KUKA KRL program: ps_com_geo_c1.src, ps_com_geo_c1.dat

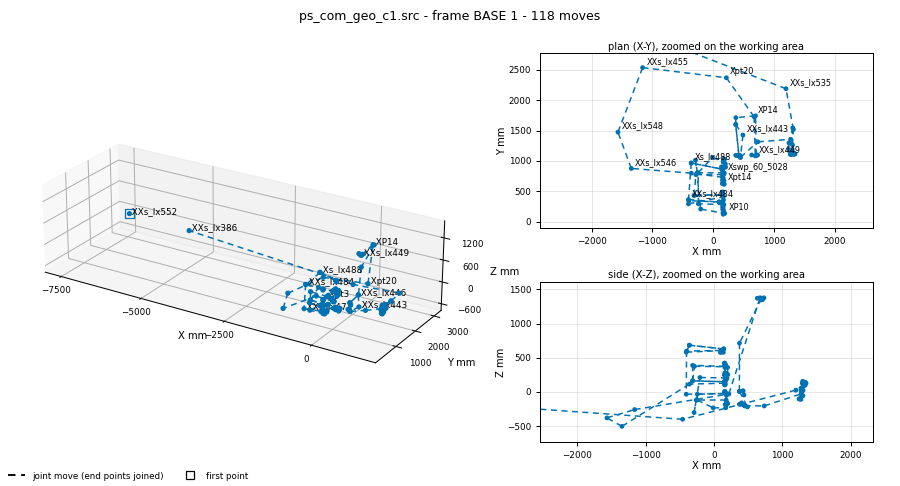
[picture p0: tool path of ps_com_geo_c1.src in frame BASE 1, 118 of 121 moves have a stored position in this frame; points joined in program order, loops and branches not executed]
--- ps_com_geo_c1.src ---
&ACCESS RVO1
&REL 24
&COMMENT Solda GUN C1 Geometria
&PARAM DISKPATH = KRC:\R1\Program\SOLDA LTC
DEF ps_com_geo_c1( )
;FOLD INI
;FOLD SPOTTECH INI
USERSPOT(#INIT)
;ENDFOLD (SPOTTECH INI)
  ;FOLD USER INI
    ;Make your modifications here

  ;ENDFOLD (USER INI)
;ENDFOLD (INI)

; Caracterização dos meios de produção:
; Versão Atual:
; 15/07/2013 12:00 Name: P13.050-R4 CHANGES: Geometria Actros
; LTA/LTB/MGS/MGSB/STB Pinça C1

chk_w1_wechs_ok ( )     ; CHECK FERRAMENTA: C1

;FOLD PTP Xs_lx552 CONT Vel=100 % PDAT57 Tool[1]:GUN_C1 Base[1]:ACTROS;%{PE}%R 8.2.20,%MKUKATPBASIS,%CMOVE,%VPTP,%P 1:PTP, 2:Xs_lx552, 3:C_DIS, 5:100, 7:PDAT57
$BWDSTART=FALSE
PDAT_ACT=PPDAT57
FDAT_ACT=FXs_lx552
BAS(#PTP_PARAMS,100)
PTP XXs_lx552 C_DIS
;ENDFOLD

if MaxStandMenge (1) then
  MaxStandmengeErreicht (1)
endif

IF (NOT(GHOST())) THEN
if Elektrodenwechsel (1) then
  e_Fraes1 ()
endif
ENDIF

;FOLD PTP c_lx33 CONT Vel=100 % P_OLP116 Tool[1]:GUN_C1 Base[1]:ACTROS;%{PE}%R 8.2.20,%MKUKATPBASIS,%CMOVE,%VPTP,%P 1:PTP, 2:c_lx33, 3:C_DIS, 5:100, 7:P_OLP116
$BWDSTART=FALSE
PDAT_ACT=PP_OLP116
FDAT_ACT=Fc_lx33
BAS(#PTP_PARAMS,100)
PTP Xc_lx33 C_DIS
;ENDFOLD
;FOLD PTP P3 CONT Vel=100 % PDAT59 Tool[1]:GUN_C1 Base[1]:ACTROS;%{PE}%R 8.2.20,%MKUKATPBASIS,%CMOVE,%VPTP,%P 1:PTP, 2:P3, 3:C_DIS, 5:100, 7:PDAT59
$BWDSTART=FALSE
PDAT_ACT=PPDAT59
FDAT_ACT=FP3
BAS(#PTP_PARAMS,100)
PTP XP3 C_DIS
;ENDFOLD
;FOLD PTP P2 Vel=100 % PDAT58 Tool[8]:TOOL_CHANGE Base[0];%{PE}%R 8.2.20,%MKUKATPBASIS,%CMOVE,%VPTP,%P 1:PTP, 2:P2, 3:, 5:100, 7:PDAT58
$BWDSTART=FALSE
PDAT_ACT=PPDAT58
FDAT_ACT=FP2
BAS(#PTP_PARAMS,100)
PTP XP2
;ENDFOLD

;FOLD OUT 3339 'R4 soldando' State=TRUE ;%{PE}%R 8.2.20,%MKUKATPBASIS,%COUT,%VOUTX,%P 2:3339, 3:R4 soldando, 5:TRUE, 6:
$OUT[3339]=TRUE
;ENDFOLD
;FOLD WAIT FOR ( IN 3339 'Aguarda lib solsar geometria' );%{PE}%R 8.2.20,%MKUKATPBASIS,%CEXT_WAIT_FOR,%VEXT_WAIT_FOR,%P 2:, 4:, 5:$IN, 6:3339, 7:Aguarda lib solsar geometria, 9:
WAIT FOR  ( $IN[3339] )
;ENDFOLD
;FOLD OUT 3339 'R4 soldando' State=FALSE ;%{PE}%R 8.2.20,%MKUKATPBASIS,%COUT,%VOUTX,%P 2:3339, 3:R4 soldando, 5:FALSE, 6:
$OUT[3339]=FALSE
;ENDFOLD
;FOLD OUT 3343 'R4 entregou peca Geo' State=FALSE ;%{PE}%R 8.2.20,%MKUKATPBASIS,%COUT,%VOUTX,%P 2:3343, 3:R4 entregou peca Geo, 5:FALSE, 6:
$OUT[3343]=FALSE
;ENDFOLD
;FOLD OUT 3348 'Fora area GEOBOX' State=FALSE ;%{PE}%R 8.2.20,%MKUKATPBASIS,%COUT,%VOUTX,%P 2:3348, 3:Fora area GEOBOX, 5:FALSE, 6:
$OUT[3348]=FALSE
;ENDFOLD
;FOLD  ;%{PE}%R 8.2.20,%MKUKATPBASIS,%CCOMMENT,%VNORMAL,%P 2:
;ENDFOLD
;FOLD Collision.Monitoring_5_On ;%{PE}%MKUKATPUSER
COLLSTOP( 5, 1 ) ;not Interrupt-Controlled
;ENDFOLD

;FOLD PTP Xs_lx488 CONT Vel=100 % P_OLP5 Tool[1]:GUN_C1 Base[1]:ACTROS;%{PE}%R8.2,%MKUKATPBASIS,%CMOVE,%VPTP,%P 1:PTP, 2:Xs_lx488, 3:C_DIS, 5:100, 7:P_OLP5
$BWDSTART = FALSE
PDAT_ACT= PP_OLP5
FDAT_ACT= Fs_lx488
BAS(#PTP_PARAMS,100)
PTP Xs_lx488 C_DIS
;ENDFOLD
;FOLD PTP Xs_lx487 CONT Vel=100 % PDAT2 Tool[1]:GUN_C1 Base[1]:ACTROS;%{PE}%R 8.2.19,%MKUKATPBASIS,%CMOVE,%VPTP,%P 1:PTP, 2:Xs_lx487, 3:C_DIS, 5:100, 7:PDAT2
$BWDSTART=FALSE
PDAT_ACT=PPDAT2
FDAT_ACT=FXs_lx487
BAS(#PTP_PARAMS,100)
PTP XXs_lx487 C_DIS
;ENDFOLD

;FOLD ; swp_60_5140;%{PE}%R 5.4.33,%MKUKATPBASIS,%CCOMMENT,%VNORMAL,%P 2:swp_60_5140
;ENDFOLD
;FOLD PTP swp_60_5140 P_OLP7 SPOT Gun=1 RETR CLS PgNo1=14 ACTIVE=1 Tool[1]:GUN_C1 Base[1]:ACTROS;%{PE}%R 8.2.2,%MKUKATPSPOT,%CSPOT,%VPTP,%P 1:PTP, 2:swp_60_5140, 3:, 5:100, 7:P_OLP7, 10:1, 12:#FIRST, 14:#CLO, 16:14, 18:1, 20:1, 22:0, 24:1, 25:S_OLP1
$BWDSTART=FALSE
PDAT_ACT=PP_OLP7
FDAT_ACT=Fswp_60_5140
BAS(#PTP_PARAMS,PP_OLP7.VEL)
S_ACT.GUN=1
S_ACT.PAIR=SDEFAULT.PAIR
S_ACT.RETR=#CLO
S_ACT.CLO_TM=1
S_ACT.PGNO1=14
S_ACT.PGNO2=SDEFAULT.PGNO2
S_ACT.PRESS1=SDEFAULT.PRESS1
S_ACT.PRESS2=SDEFAULT.PRESS2
S_READY=FALSE
PTP Xswp_60_5140
USERSPOT(#SPOT, S_ACT)
WAIT FOR S_READY
;ENDFOLD

;FOLD PTP Xs_lx502 CONT Vel=100 % PDAT6 Tool[1]:GUN_C1 Base[1]:ACTROS;%{PE}%R 8.2.20,%MKUKATPBASIS,%CMOVE,%VPTP,%P 1:PTP, 2:Xs_lx502, 3:C_DIS, 5:100, 7:PDAT6
$BWDSTART=FALSE
PDAT_ACT=PPDAT6
FDAT_ACT=FXs_lx502
BAS(#PTP_PARAMS,100)
PTP XXs_lx502 C_DIS
;ENDFOLD
;FOLD PTP Xs_lx486 CONT Vel=100 % P_OLP9 Tool[1]:GUN_C1 Base[1]:ACTROS;%{PE}%R8.2,%MKUKATPBASIS,%CMOVE,%VPTP,%P 1:PTP, 2:Xs_lx486, 3:C_DIS, 5:100, 7:P_OLP9
$BWDSTART = FALSE
PDAT_ACT= PP_OLP9
FDAT_ACT= Fs_lx486
BAS(#PTP_PARAMS,100)
PTP Xs_lx486 C_DIS
;ENDFOLD
;FOLD  ;%{PE}%R 8.2.20,%MKUKATPBASIS,%CCOMMENT,%VNORMAL,%P 2:
;ENDFOLD
;FOLD Collision.Monitoring_5_Off . ;%{PE}%MKUKATPUSER
COLLSTOP( 5, 2+0 )
;ENDFOLD

;FOLD PTP Xs_lx484 CONT Vel=100 % P_OLP10 Tool[1]:GUN_C1 Base[1]:ACTROS;%{PE}%R 8.2.20,%MKUKATPBASIS,%CMOVE,%VPTP,%P 1:PTP, 2:Xs_lx484, 3:C_DIS, 5:100, 7:P_OLP10
$BWDSTART=FALSE
PDAT_ACT=PP_OLP10
FDAT_ACT=FXs_lx484
BAS(#PTP_PARAMS,100)
PTP XXs_lx484 C_DIS
;ENDFOLD
;FOLD PTP Xs_lx504 CONT Vel=100 % PDAT8 Tool[1]:GUN_C1 Base[1]:ACTROS;%{PE}%R 8.2.20,%MKUKATPBASIS,%CMOVE,%VPTP,%P 1:PTP, 2:Xs_lx504, 3:C_DIS, 5:100, 7:PDAT8
$BWDSTART=FALSE
PDAT_ACT=PPDAT8
FDAT_ACT=FXs_lx504
BAS(#PTP_PARAMS,100)
PTP XXs_lx504 C_DIS
;ENDFOLD

;FOLD ; swp_60_5118;%{PE}%R 5.4.33,%MKUKATPBASIS,%CCOMMENT,%VNORMAL,%P 2:swp_60_5118
;ENDFOLD
;FOLD PTP swp_60_5118 P_OLP12 SPOT Gun=1 RETR CLS PgNo1=15 ACTIVE=1 Tool[1]:GUN_C1 Base[1]:ACTROS;%{PE}%R 8.2.2,%MKUKATPSPOT,%CSPOT,%VPTP,%P 1:PTP, 2:swp_60_5118, 3:, 5:100, 7:P_OLP12, 10:1, 12:#FIRST, 14:#CLO, 16:15, 18:1, 20:1, 22:0, 24:1, 25:S_OLP2
$BWDSTART=FALSE
PDAT_ACT=PP_OLP12
FDAT_ACT=Fswp_60_5118
BAS(#PTP_PARAMS,PP_OLP12.VEL)
S_ACT.GUN=1
S_ACT.PAIR=SDEFAULT.PAIR
S_ACT.RETR=#CLO
S_ACT.CLO_TM=1
S_ACT.PGNO1=15
S_ACT.PGNO2=SDEFAULT.PGNO2
S_ACT.PRESS1=SDEFAULT.PRESS1
S_ACT.PRESS2=SDEFAULT.PRESS2
S_READY=FALSE
PTP Xswp_60_5118
USERSPOT(#SPOT, S_ACT)
WAIT FOR S_READY
;ENDFOLD

;FOLD PTP Xs_lx506 CONT Vel=100 % PDAT10 Tool[1]:GUN_C1 Base[1]:ACTROS;%{PE}%R 8.2.20,%MKUKATPBASIS,%CMOVE,%VPTP,%P 1:PTP, 2:Xs_lx506, 3:C_DIS, 5:100, 7:PDAT10
$BWDSTART=FALSE
PDAT_ACT=PPDAT10
FDAT_ACT=FXs_lx506
BAS(#PTP_PARAMS,100)
PTP XXs_lx506 C_DIS
;ENDFOLD
;FOLD PTP Xs_lx482 CONT Vel=100 % P_OLP14 Tool[1]:GUN_C1 Base[1]:ACTROS;%{PE}%R 8.2.20,%MKUKATPBASIS,%CMOVE,%VPTP,%P 1:PTP, 2:Xs_lx482, 3:C_DIS, 5:100, 7:P_OLP14
$BWDSTART=FALSE
PDAT_ACT=PP_OLP14
FDAT_ACT=FXs_lx482
BAS(#PTP_PARAMS,100)
PTP XXs_lx482 C_DIS
;ENDFOLD
;FOLD PTP Xs_lx472 CONT Vel=100 % P_OLP16 Tool[1]:GUN_C1 Base[1]:ACTROS;%{PE}%R 8.2.20,%MKUKATPBASIS,%CMOVE,%VPTP,%P 1:PTP, 2:Xs_lx472, 3:C_DIS, 5:100, 7:P_OLP16
$BWDSTART=FALSE
PDAT_ACT=PP_OLP16
FDAT_ACT=FXs_lx472
BAS(#PTP_PARAMS,100)
PTP XXs_lx472 C_DIS
;ENDFOLD

;FOLD Collision.Monitoring_3_On ;%{PE}%MKUKATPUSER
COLLSTOP( 3, 1 ) ;Interrupt-Controlled
;ENDFOLD

;FOLD PTP Xs_lx510 CONT Vel=100 % PDAT14 Tool[1]:GUN_C1 Base[1]:ACTROS;%{PE}%R 8.2.20,%MKUKATPBASIS,%CMOVE,%VPTP,%P 1:PTP, 2:Xs_lx510, 3:C_DIS, 5:100, 7:PDAT14
$BWDSTART=FALSE
PDAT_ACT=PPDAT14
FDAT_ACT=FXs_lx510
BAS(#PTP_PARAMS,100)
PTP XXs_lx510 C_DIS
;ENDFOLD

;FOLD ; swp_60_5026;%{PE}%R 5.4.33,%MKUKATPBASIS,%CCOMMENT,%VNORMAL,%P 2:swp_60_5026
;ENDFOLD
;FOLD PTP swp_60_5026 P_OLP18 SPOT Gun=1 RETR CLS PgNo1=16 ACTIVE=1 Tool[1]:GUN_C1 Base[1]:ACTROS;%{PE}%R 8.2.2,%MKUKATPSPOT,%CSPOT,%VPTP,%P 1:PTP, 2:swp_60_5026, 3:, 5:100, 7:P_OLP18, 10:1, 12:#FIRST, 14:#CLO, 16:16, 18:1, 20:1, 22:0, 24:1, 25:S_OLP3
$BWDSTART=FALSE
PDAT_ACT=PP_OLP18
FDAT_ACT=Fswp_60_5026
BAS(#PTP_PARAMS,PP_OLP18.VEL)
S_ACT.GUN=1
S_ACT.PAIR=SDEFAULT.PAIR
S_ACT.RETR=#CLO
S_ACT.CLO_TM=1
S_ACT.PGNO1=16
S_ACT.PGNO2=SDEFAULT.PGNO2
S_ACT.PRESS1=SDEFAULT.PRESS1
S_ACT.PRESS2=SDEFAULT.PRESS2
S_READY=FALSE
PTP Xswp_60_5026
USERSPOT(#SPOT, S_ACT)
WAIT FOR S_READY
;ENDFOLD

;FOLD ; swp_60_5020;%{PE}%R 5.4.33,%MKUKATPBASIS,%CCOMMENT,%VNORMAL,%P 2:swp_60_5020
;ENDFOLD
;FOLD PTP swp_60_5020 P_OLP19 SPOT Gun=1 RETR CLS PgNo1=17 ACTIVE=1 Tool[1]:GUN_C1 Base[1]:ACTROS;%{PE}%R 8.2.2,%MKUKATPSPOT,%CSPOT,%VPTP,%P 1:PTP, 2:swp_60_5020, 3:, 5:100, 7:P_OLP19, 10:1, 12:#FIRST, 14:#CLO, 16:17, 18:1, 20:1, 22:0, 24:1, 25:S_OLP4
$BWDSTART=FALSE
PDAT_ACT=PP_OLP19
FDAT_ACT=Fswp_60_5020
BAS(#PTP_PARAMS,PP_OLP19.VEL)
S_ACT.GUN=1
S_ACT.PAIR=SDEFAULT.PAIR
S_ACT.RETR=#CLO
S_ACT.CLO_TM=1
S_ACT.PGNO1=17
S_ACT.PGNO2=SDEFAULT.PGNO2
S_ACT.PRESS1=SDEFAULT.PRESS1
S_ACT.PRESS2=SDEFAULT.PRESS2
S_READY=FALSE
PTP Xswp_60_5020
USERSPOT(#SPOT, S_ACT)
WAIT FOR S_READY
;ENDFOLD

;FOLD ; swp_60_5016;%{PE}%R 5.4.33,%MKUKATPBASIS,%CCOMMENT,%VNORMAL,%P 2:swp_60_5016
;ENDFOLD
;FOLD PTP swp_60_5016 P_OLP20 SPOT Gun=1 RETR CLS PgNo1=18 ACTIVE=1 Tool[1]:GUN_C1 Base[1]:ACTROS;%{PE}%R 8.2.2,%MKUKATPSPOT,%CSPOT,%VPTP,%P 1:PTP, 2:swp_60_5016, 3:, 5:100, 7:P_OLP20, 10:1, 12:#FIRST, 14:#CLO, 16:18, 18:1, 20:1, 22:0, 24:1, 25:S_OLP5
$BWDSTART=FALSE
PDAT_ACT=PP_OLP20
FDAT_ACT=Fswp_60_5016
BAS(#PTP_PARAMS,PP_OLP20.VEL)
S_ACT.GUN=1
S_ACT.PAIR=SDEFAULT.PAIR
S_ACT.RETR=#CLO
S_ACT.CLO_TM=1
S_ACT.PGNO1=18
S_ACT.PGNO2=SDEFAULT.PGNO2
S_ACT.PRESS1=SDEFAULT.PRESS1
S_ACT.PRESS2=SDEFAULT.PRESS2
S_READY=FALSE
PTP Xswp_60_5016
USERSPOT(#SPOT, S_ACT)
WAIT FOR S_READY
;ENDFOLD

;FOLD ; swp_60_5014;%{PE}%R 5.4.33,%MKUKATPBASIS,%CCOMMENT,%VNORMAL,%P 2:swp_60_5014
;ENDFOLD
;FOLD PTP swp_60_5014 P_OLP21 SPOT Gun=1 RETR CLS PgNo1=19 ACTIVE=1 Tool[1]:GUN_C1 Base[1]:ACTROS;%{PE}%R 8.2.2,%MKUKATPSPOT,%CSPOT,%VPTP,%P 1:PTP, 2:swp_60_5014, 3:, 5:100, 7:P_OLP21, 10:1, 12:#FIRST, 14:#CLO, 16:19, 18:1, 20:1, 22:0, 24:1, 25:S_OLP6
$BWDSTART=FALSE
PDAT_ACT=PP_OLP21
FDAT_ACT=Fswp_60_5014
BAS(#PTP_PARAMS,PP_OLP21.VEL)
S_ACT.GUN=1
S_ACT.PAIR=SDEFAULT.PAIR
S_ACT.RETR=#CLO
S_ACT.CLO_TM=1
S_ACT.PGNO1=19
S_ACT.PGNO2=SDEFAULT.PGNO2
S_ACT.PRESS1=SDEFAULT.PRESS1
S_ACT.PRESS2=SDEFAULT.PRESS2
S_READY=FALSE
PTP Xswp_60_5014
USERSPOT(#SPOT, S_ACT)
WAIT FOR S_READY
;ENDFOLD

;FOLD PTP Xs_lx469 CONT Vel=100 % P_OLP22 Tool[1]:GUN_C1 Base[1]:ACTROS;%{PE}%R 8.2.19,%MKUKATPBASIS,%CMOVE,%VPTP,%P 1:PTP, 2:Xs_lx469, 3:C_DIS, 5:100, 7:P_OLP22
$BWDSTART=FALSE
PDAT_ACT=PP_OLP22
FDAT_ACT=FXs_lx469
BAS(#PTP_PARAMS,100)
PTP XXs_lx469 C_DIS
;ENDFOLD
;FOLD PTP Xs_lx470 CONT Vel=100 % P_OLP23 Tool[1]:GUN_C1 Base[1]:ACTROS;%{PE}%R8.2,%MKUKATPBASIS,%CMOVE,%VPTP,%P 1:PTP, 2:Xs_lx470, 3:C_DIS, 5:100, 7:P_OLP23
$BWDSTART = FALSE
PDAT_ACT= PP_OLP23
FDAT_ACT= Fs_lx470
BAS(#PTP_PARAMS,100)
PTP Xs_lx470 C_DIS
;ENDFOLD
;FOLD PTP Xs_lx468 Vel=100 % P_OLP24 Tool[1]:GUN_C1 Base[1]:ACTROS;%{PE}%R 8.2.20,%MKUKATPBASIS,%CMOVE,%VPTP,%P 1:PTP, 2:Xs_lx468, 3:, 5:100, 7:P_OLP24
$BWDSTART=FALSE
PDAT_ACT=PP_OLP24
FDAT_ACT=FXs_lx468
BAS(#PTP_PARAMS,100)
PTP XXs_lx468
;ENDFOLD

;FOLD Collision.Monitoring_3_Off . ;%{PE}%MKUKATPUSER
COLLSTOP( 3, 2+0 )
;ENDFOLD
;FOLD ;%{PE}%R 8.2.20,%MKUKATPBASIS,%CCOMMENT,%VNORMAL,%P 2:
;ENDFOLD
;FOLD PTP Xlx507 CONT Vel=100 % P_OLP25 Tool[1]:GUN_C1 Base[1]:ACTROS;%{PE}%R8.2,%MKUKATPBASIS,%CMOVE,%VPTP,%P 1:PTP, 2:Xlx507, 3:C_DIS, 5:100, 7:P_OLP25
$BWDSTART = FALSE
PDAT_ACT= PP_OLP25
FDAT_ACT= Flx507
BAS(#PTP_PARAMS,100)
PTP Xlx507 C_DIS
;ENDFOLD
;FOLD PTP Xs_lx467 CONT Vel=100 % P_OLP26 Tool[1]:GUN_C1 Base[1]:ACTROS;%{PE}%R 8.2.20,%MKUKATPBASIS,%CMOVE,%VPTP,%P 1:PTP, 2:Xs_lx467, 3:C_DIS, 5:100, 7:P_OLP26
$BWDSTART=FALSE
PDAT_ACT=PP_OLP26
FDAT_ACT=FXs_lx467
BAS(#PTP_PARAMS,100)
PTP XXs_lx467 C_DIS
;ENDFOLD

;FOLD ; swp_60_5042;%{PE}%R 5.4.33,%MKUKATPBASIS,%CCOMMENT,%VNORMAL,%P 2:swp_60_5042
;ENDFOLD
;FOLD PTP swp_60_5042 P_OLP27 SPOT Gun=1 RETR CLS PgNo1=20 ACTIVE=1 Tool[1]:GUN_C1 Base[1]:ACTROS;%{PE}%R 8.2.2,%MKUKATPSPOT,%CSPOT,%VPTP,%P 1:PTP, 2:swp_60_5042, 3:, 5:100, 7:P_OLP27, 10:1, 12:#FIRST, 14:#CLO, 16:20, 18:1, 20:1, 22:0, 24:1, 25:S_OLP7
$BWDSTART=FALSE
PDAT_ACT=PP_OLP27
FDAT_ACT=Fswp_60_5042
BAS(#PTP_PARAMS,PP_OLP27.VEL)
S_ACT.GUN=1
S_ACT.PAIR=SDEFAULT.PAIR
S_ACT.RETR=#CLO
S_ACT.CLO_TM=1
S_ACT.PGNO1=20
S_ACT.PGNO2=SDEFAULT.PGNO2
S_ACT.PRESS1=SDEFAULT.PRESS1
S_ACT.PRESS2=SDEFAULT.PRESS2
S_READY=FALSE
PTP Xswp_60_5042
USERSPOT(#SPOT, S_ACT)
WAIT FOR S_READY
;ENDFOLD

;FOLD PTP Xs_lx512 CONT Vel=100 % PDAT16 Tool[1]:GUN_C1 Base[1]:ACTROS;%{PE}%R 8.2.19,%MKUKATPBASIS,%CMOVE,%VPTP,%P 1:PTP, 2:Xs_lx512, 3:C_DIS, 5:100, 7:PDAT16
$BWDSTART=FALSE
PDAT_ACT=PPDAT16
FDAT_ACT=FXs_lx512
BAS(#PTP_PARAMS,100)
PTP XXs_lx512 C_DIS
;ENDFOLD

;FOLD ; swp_60_5040;%{PE}%R 5.4.33,%MKUKATPBASIS,%CCOMMENT,%VNORMAL,%P 2:swp_60_5040
;ENDFOLD
;FOLD PTP swp_60_5040 P_OLP28 SPOT Gun=1 RETR CLS PgNo1=21 ACTIVE=1 Tool[1]:GUN_C1 Base[1]:ACTROS;%{PE}%R 8.2.2,%MKUKATPSPOT,%CSPOT,%VPTP,%P 1:PTP, 2:swp_60_5040, 3:, 5:100, 7:P_OLP28, 10:1, 12:#FIRST, 14:#CLO, 16:21, 18:1, 20:1, 22:0, 24:1, 25:S_OLP8
$BWDSTART=FALSE
PDAT_ACT=PP_OLP28
FDAT_ACT=Fswp_60_5040
BAS(#PTP_PARAMS,PP_OLP28.VEL)
S_ACT.GUN=1
S_ACT.PAIR=SDEFAULT.PAIR
S_ACT.RETR=#CLO
S_ACT.CLO_TM=1
S_ACT.PGNO1=21
S_ACT.PGNO2=SDEFAULT.PGNO2
S_ACT.PRESS1=SDEFAULT.PRESS1
S_ACT.PRESS2=SDEFAULT.PRESS2
S_READY=FALSE
PTP Xswp_60_5040
USERSPOT(#SPOT, S_ACT)
WAIT FOR S_READY
;ENDFOLD

;FOLD ; swp_60_5038;%{PE}%R 5.4.33,%MKUKATPBASIS,%CCOMMENT,%VNORMAL,%P 2:swp_60_5038
;ENDFOLD
;FOLD PTP swp_60_5038 P_OLP29 SPOT Gun=1 RETR OPN PgNo1=22 ACTIVE=1 Tool[1]:GUN_C1 Base[1]:ACTROS;%{PE}%R 8.2.2,%MKUKATPSPOT,%CSPOT,%VPTP,%P 1:PTP, 2:swp_60_5038, 3:, 5:100, 7:P_OLP29, 10:1, 12:#FIRST, 14:#OPN, 16:22, 18:1, 20:1, 22:0, 24:1, 25:S_OLP9
$BWDSTART=FALSE
PDAT_ACT=PP_OLP29
FDAT_ACT=Fswp_60_5038
BAS(#PTP_PARAMS,PP_OLP29.VEL)
S_ACT.GUN=1
S_ACT.PAIR=SDEFAULT.PAIR
S_ACT.RETR=#OPN
S_ACT.CLO_TM=1
S_ACT.PGNO1=22
S_ACT.PGNO2=SDEFAULT.PGNO2
S_ACT.PRESS1=SDEFAULT.PRESS1
S_ACT.PRESS2=SDEFAULT.PRESS2
S_READY=FALSE
PTP Xswp_60_5038
USERSPOT(#SPOT, S_ACT)
WAIT FOR S_READY
;ENDFOLD

;FOLD PTP Xs_lx514 CONT Vel=100 % PDAT18 Tool[1]:GUN_C1 Base[1]:ACTROS;%{PE}%R 8.2.19,%MKUKATPBASIS,%CMOVE,%VPTP,%P 1:PTP, 2:Xs_lx514, 3:C_DIS, 5:100, 7:PDAT18
$BWDSTART=FALSE
PDAT_ACT=PPDAT18
FDAT_ACT=FXs_lx514
BAS(#PTP_PARAMS,100)
PTP XXs_lx514 C_DIS
;ENDFOLD

;FOLD ; swp_60_5036;%{PE}%R 5.4.33,%MKUKATPBASIS,%CCOMMENT,%VNORMAL,%P 2:swp_60_5036
;ENDFOLD
;FOLD PTP swp_60_5036 PDAT45 SPOT Gun=1 RETR CLS PgNo1=23 ACTIVE=1 Tool[1]:GUN_C1 Base[1]:ACTROS;%{PE}%R 8.2.2,%MKUKATPSPOT,%CSPOT,%VPTP,%P 1:PTP, 2:swp_60_5036, 3:, 5:100, 7:PDAT45, 10:1, 12:#FIRST, 14:#CLO, 16:23, 18:1, 20:1, 22:0, 24:1, 25:S_OLP10
$BWDSTART=FALSE
PDAT_ACT=PPDAT45
FDAT_ACT=Fswp_60_5036
BAS(#PTP_PARAMS,PPDAT45.VEL)
S_ACT.GUN=1
S_ACT.PAIR=SDEFAULT.PAIR
S_ACT.RETR=#CLO
S_ACT.CLO_TM=1
S_ACT.PGNO1=23
S_ACT.PGNO2=SDEFAULT.PGNO2
S_ACT.PRESS1=SDEFAULT.PRESS1
S_ACT.PRESS2=SDEFAULT.PRESS2
S_READY=FALSE
PTP Xswp_60_5036
USERSPOT(#SPOT, S_ACT)
WAIT FOR S_READY
;ENDFOLD

;FOLD ; swp_60_5028;%{PE}%R 8.2.20,%MKUKATPBASIS,%CCOMMENT,%VNORMAL,%P 2:swp_60_5028
;ENDFOLD
;FOLD PTP swp_60_5028 P_OLP32 SPOT Gun=1 RETR CLS PgNo1=24 ACTIVE=1 Tool[1]:GUN_C1 Base[1]:ACTROS;%{PE}%R 8.2.2,%MKUKATPSPOT,%CSPOT,%VPTP,%P 1:PTP, 2:swp_60_5028, 3:, 5:100, 7:P_OLP32, 10:1, 12:#FIRST, 14:#CLO, 16:24, 18:1, 20:1, 22:0, 24:1, 25:S_OLP11
$BWDSTART=FALSE
PDAT_ACT=PP_OLP32
FDAT_ACT=Fswp_60_5028
BAS(#PTP_PARAMS,PP_OLP32.VEL)
S_ACT.GUN=1
S_ACT.PAIR=SDEFAULT.PAIR
S_ACT.RETR=#CLO
S_ACT.CLO_TM=1
S_ACT.PGNO1=24
S_ACT.PGNO2=SDEFAULT.PGNO2
S_ACT.PRESS1=SDEFAULT.PRESS1
S_ACT.PRESS2=SDEFAULT.PRESS2
S_READY=FALSE
PTP Xswp_60_5028
USERSPOT(#SPOT, S_ACT)
WAIT FOR S_READY
;ENDFOLD

;FOLD PTP Xs_lx464 CONT Vel=100 % P_OLP33 Tool[1]:GUN_C1 Base[1]:ACTROS;%{PE}%R8.2,%MKUKATPBASIS,%CMOVE,%VPTP,%P 1:PTP, 2:Xs_lx464, 3:C_DIS, 5:100, 7:P_OLP33
$BWDSTART = FALSE
PDAT_ACT= PP_OLP33
FDAT_ACT= Fs_lx464
BAS(#PTP_PARAMS,100)
PTP Xs_lx464 C_DIS
;ENDFOLD
;FOLD PTP Xs_lx465 CONT Vel=100 % P_OLP34 Tool[1]:GUN_C1 Base[1]:ACTROS;%{PE}%R 8.2.19,%MKUKATPBASIS,%CMOVE,%VPTP,%P 1:PTP, 2:Xs_lx465, 3:C_DIS, 5:100, 7:P_OLP34
$BWDSTART=FALSE
PDAT_ACT=PP_OLP34
FDAT_ACT=FXs_lx465
BAS(#PTP_PARAMS,100)
PTP XXs_lx465 C_DIS
;ENDFOLD
;FOLD PTP P8 CONT Vel=100 % PDAT65 Tool[1]:GUN_C1 Base[1]:ACTROS;%{PE}%R 8.2.20,%MKUKATPBASIS,%CMOVE,%VPTP,%P 1:PTP, 2:P8, 3:C_DIS, 5:100, 7:PDAT65
$BWDSTART=FALSE
PDAT_ACT=PPDAT65
FDAT_ACT=FP8
BAS(#PTP_PARAMS,100)
PTP XP8 C_DIS
;ENDFOLD
;FOLD ;%{PE}%R 8.2.20,%MKUKATPBASIS,%CCOMMENT,%VNORMAL,%P 2:
;ENDFOLD
;FOLD Collision.Monitoring_AREA_6_On ;%{PE}%MKUKATPUSER
COLLSTOP( 12, 1 ) ;not Interrupt-Controlled
;ENDFOLD
;FOLD ;%{PE}%R 8.2.20,%MKUKATPBASIS,%CCOMMENT,%VNORMAL,%P 2:
;ENDFOLD
;FOLD PTP P9 CONT Vel=100 % PDAT66 Tool[1]:GUN_C1 Base[1]:ACTROS;%{PE}%R 8.2.20,%MKUKATPBASIS,%CMOVE,%VPTP,%P 1:PTP, 2:P9, 3:C_DIS, 5:100, 7:PDAT66
$BWDSTART=FALSE
PDAT_ACT=PPDAT66
FDAT_ACT=FP9
BAS(#PTP_PARAMS,100)
PTP XP9 C_DIS
;ENDFOLD
;FOLD PTP P10 CONT Vel=100 % PDAT67 Tool[1]:GUN_C1 Base[1]:ACTROS;%{PE}%R 8.2.20,%MKUKATPBASIS,%CMOVE,%VPTP,%P 1:PTP, 2:P10, 3:C_DIS, 5:100, 7:PDAT67
$BWDSTART=FALSE
PDAT_ACT=PPDAT67
FDAT_ACT=FP10
BAS(#PTP_PARAMS,100)
PTP XP10 C_DIS
;ENDFOLD

;FOLD ; swp_60_5218;%{PE}%R 8.2.20,%MKUKATPBASIS,%CCOMMENT,%VNORMAL,%P 2:swp_60_5218
;ENDFOLD
;FOLD PTP swp_60_5218 PDAT68 SPOT Gun=1 RETR CLS PgNo1=29 ACTIVE=1 Tool[1]:GUN_C1 Base[1]:ACTROS;%{PE}%R 8.2.2,%MKUKATPSPOT,%CSPOT,%VPTP,%P 1:PTP, 2:swp_60_5218, 3:, 5:100, 7:PDAT68, 10:1, 12:#FIRST, 14:#CLO, 16:29, 18:1, 20:0, 22:0, 24:1, 25:NORMAL
$BWDSTART=FALSE
PDAT_ACT=PPDAT68
FDAT_ACT=Fswp_60_5218
BAS(#PTP_PARAMS,PPDAT68.VEL)
S_ACT.GUN=1
S_ACT.PAIR=SDEFAULT.PAIR
S_ACT.RETR=#CLO
S_ACT.CLO_TM=1
S_ACT.PGNO1=29
S_ACT.PGNO2=SDEFAULT.PGNO2
S_ACT.PRESS1=SDEFAULT.PRESS1
S_ACT.PRESS2=SDEFAULT.PRESS2
S_READY=FALSE
PTP Xswp_60_5218
USERSPOT(#SPOT, S_ACT)
WAIT FOR S_READY
;ENDFOLD

;FOLD PTP P13 CONT Vel=100 % PDAT70 Tool[1]:GUN_C1 Base[1]:ACTROS;%{PE}%R 8.2.20,%MKUKATPBASIS,%CMOVE,%VPTP,%P 1:PTP, 2:P13, 3:C_DIS, 5:100, 7:PDAT70
$BWDSTART=FALSE
PDAT_ACT=PPDAT70
FDAT_ACT=FP13
BAS(#PTP_PARAMS,100)
PTP XP13 C_DIS
;ENDFOLD

;FOLD ; swp_60_5190;%{PE}%R 8.2.20,%MKUKATPBASIS,%CCOMMENT,%VNORMAL,%P 2:swp_60_5190
;ENDFOLD
;FOLD PTP swp_60_5190 PDAT71 SPOT Gun=1 RETR CLS PgNo1=28 ACTIVE=1 Tool[1]:GUN_C1 Base[1]:ACTROS;%{PE}%R 8.2.2,%MKUKATPSPOT,%CSPOT,%VPTP,%P 1:PTP, 2:swp_60_5190, 3:, 5:100, 7:PDAT71, 10:1, 12:#FIRST, 14:#CLO, 16:28, 18:1, 20:0, 22:0, 24:1, 25:NORMAL
$BWDSTART=FALSE
PDAT_ACT=PPDAT71
FDAT_ACT=Fswp_60_5190
BAS(#PTP_PARAMS,PPDAT71.VEL)
S_ACT.GUN=1
S_ACT.PAIR=SDEFAULT.PAIR
S_ACT.RETR=#CLO
S_ACT.CLO_TM=1
S_ACT.PGNO1=28
S_ACT.PGNO2=SDEFAULT.PGNO2
S_ACT.PRESS1=SDEFAULT.PRESS1
S_ACT.PRESS2=SDEFAULT.PRESS2
S_READY=FALSE
PTP Xswp_60_5190
USERSPOT(#SPOT, S_ACT)
WAIT FOR S_READY
;ENDFOLD

;FOLD PTP pt1 CONT Vel=100 % PDAT72 Tool[1]:GUN_C1 Base[1]:ACTROS;%{PE}%R 8.2.20,%MKUKATPBASIS,%CMOVE,%VPTP,%P 1:PTP, 2:pt1, 3:C_DIS, 5:100, 7:PDAT72
$BWDSTART=FALSE
PDAT_ACT=PPDAT72
FDAT_ACT=Fpt1
BAS(#PTP_PARAMS,100)
PTP Xpt1 C_DIS
;ENDFOLD

;FOLD ; swp_60_5195;%{PE}%R 8.2.20,%MKUKATPBASIS,%CCOMMENT,%VNORMAL,%P 2:swp_60_5195
;ENDFOLD
;FOLD PTP swp_60_5195 PDAT73 SPOT Gun=1 RETR CLS PgNo1=27 ACTIVE=1 Tool[1]:GUN_C1 Base[1]:ACTROS;%{PE}%R 8.2.2,%MKUKATPSPOT,%CSPOT,%VPTP,%P 1:PTP, 2:swp_60_5195, 3:, 5:100, 7:PDAT73, 10:1, 12:#FIRST, 14:#CLO, 16:27, 18:1, 20:0, 22:0, 24:1, 25:NORMAL
$BWDSTART=FALSE
PDAT_ACT=PPDAT73
FDAT_ACT=Fswp_60_5195
BAS(#PTP_PARAMS,PPDAT73.VEL)
S_ACT.GUN=1
S_ACT.PAIR=SDEFAULT.PAIR
S_ACT.RETR=#CLO
S_ACT.CLO_TM=1
S_ACT.PGNO1=27
S_ACT.PGNO2=SDEFAULT.PGNO2
S_ACT.PRESS1=SDEFAULT.PRESS1
S_ACT.PRESS2=SDEFAULT.PRESS2
S_READY=FALSE
PTP Xswp_60_5195
USERSPOT(#SPOT, S_ACT)
WAIT FOR S_READY
;ENDFOLD

;FOLD PTP pt2 CONT Vel=100 % PDAT74 Tool[1]:GUN_C1 Base[1]:ACTROS;%{PE}%R 8.2.20,%MKUKATPBASIS,%CMOVE,%VPTP,%P 1:PTP, 2:pt2, 3:C_DIS, 5:100, 7:PDAT74
$BWDSTART=FALSE
PDAT_ACT=PPDAT74
FDAT_ACT=Fpt2
BAS(#PTP_PARAMS,100)
PTP Xpt2 C_DIS
;ENDFOLD
;FOLD PTP pt3 CONT Vel=100 % PDAT75 Tool[1]:GUN_C1 Base[1]:ACTROS;%{PE}%R 8.2.20,%MKUKATPBASIS,%CMOVE,%VPTP,%P 1:PTP, 2:pt3, 3:C_DIS, 5:100, 7:PDAT75
$BWDSTART=FALSE
PDAT_ACT=PPDAT75
FDAT_ACT=Fpt3
BAS(#PTP_PARAMS,100)
PTP Xpt3 C_DIS
;ENDFOLD

;FOLD ; swp_60_5203;%{PE}%R 8.2.20,%MKUKATPBASIS,%CCOMMENT,%VNORMAL,%P 2:swp_60_5203
;ENDFOLD
;FOLD PTP swp_60_5203 PDAT76 SPOT Gun=1 RETR CLS PgNo1=26 ACTIVE=1 Tool[1]:GUN_C1 Base[1]:ACTROS;%{PE}%R 8.2.2,%MKUKATPSPOT,%CSPOT,%VPTP,%P 1:PTP, 2:swp_60_5203, 3:, 5:100, 7:PDAT76, 10:1, 12:#FIRST, 14:#CLO, 16:26, 18:1, 20:0, 22:0, 24:1, 25:NORMAL
$BWDSTART=FALSE
PDAT_ACT=PPDAT76
FDAT_ACT=Fswp_60_5203
BAS(#PTP_PARAMS,PPDAT76.VEL)
S_ACT.GUN=1
S_ACT.PAIR=SDEFAULT.PAIR
S_ACT.RETR=#CLO
S_ACT.CLO_TM=1
S_ACT.PGNO1=26
S_ACT.PGNO2=SDEFAULT.PGNO2
S_ACT.PRESS1=SDEFAULT.PRESS1
S_ACT.PRESS2=SDEFAULT.PRESS2
S_READY=FALSE
PTP Xswp_60_5203
USERSPOT(#SPOT, S_ACT)
WAIT FOR S_READY
;ENDFOLD

;FOLD PTP pt4 Vel=100 % PDAT77 Tool[1]:GUN_C1 Base[1]:ACTROS;%{PE}%R 8.2.20,%MKUKATPBASIS,%CMOVE,%VPTP,%P 1:PTP, 2:pt4, 3:, 5:100, 7:PDAT77
$BWDSTART=FALSE
PDAT_ACT=PPDAT77
FDAT_ACT=Fpt4
BAS(#PTP_PARAMS,100)
PTP Xpt4
;ENDFOLD
;FOLD PTP pt5 CONT Vel=100 % PDAT78 Tool[1]:GUN_C1 Base[1]:ACTROS;%{PE}%R 8.2.20,%MKUKATPBASIS,%CMOVE,%VPTP,%P 1:PTP, 2:pt5, 3:C_DIS, 5:100, 7:PDAT78
$BWDSTART=FALSE
PDAT_ACT=PPDAT78
FDAT_ACT=Fpt5
BAS(#PTP_PARAMS,100)
PTP Xpt5 C_DIS
;ENDFOLD
;FOLD PTP pt6 CONT Vel=100 % PDAT79 Tool[1]:GUN_C1 Base[1]:ACTROS;%{PE}%R 8.2.20,%MKUKATPBASIS,%CMOVE,%VPTP,%P 1:PTP, 2:pt6, 3:C_DIS, 5:100, 7:PDAT79
$BWDSTART=FALSE
PDAT_ACT=PPDAT79
FDAT_ACT=Fpt6
BAS(#PTP_PARAMS,100)
PTP Xpt6 C_DIS
;ENDFOLD
;FOLD PTP pt7 Vel=100 % PDAT80 Tool[1]:GUN_C1 Base[1]:ACTROS;%{PE}%R 8.2.20,%MKUKATPBASIS,%CMOVE,%VPTP,%P 1:PTP, 2:pt7, 3:, 5:100, 7:PDAT80
$BWDSTART=FALSE
PDAT_ACT=PPDAT80
FDAT_ACT=Fpt7
BAS(#PTP_PARAMS,100)
PTP Xpt7
;ENDFOLD

; swp_60_5209
;FOLD PTP swp_60_5209 PDAT81 SPOT Gun=1 RETR CLS PgNo1=25 ACTIVE=1 Tool[1]:GUN_C1 Base[1]:ACTROS;%{PE}%R 8.2.2,%MKUKATPSPOT,%CSPOT,%VPTP,%P 1:PTP, 2:swp_60_5209, 3:, 5:100, 7:PDAT81, 10:1, 12:#FIRST, 14:#CLO, 16:25, 18:1, 20:0, 22:0, 24:1, 25:NORMAL
$BWDSTART=FALSE
PDAT_ACT=PPDAT81
FDAT_ACT=Fswp_60_5209
BAS(#PTP_PARAMS,PPDAT81.VEL)
S_ACT.GUN=1
S_ACT.PAIR=SDEFAULT.PAIR
S_ACT.RETR=#CLO
S_ACT.CLO_TM=1
S_ACT.PGNO1=25
S_ACT.PGNO2=SDEFAULT.PGNO2
S_ACT.PRESS1=SDEFAULT.PRESS1
S_ACT.PRESS2=SDEFAULT.PRESS2
S_READY=FALSE
PTP Xswp_60_5209
USERSPOT(#SPOT, S_ACT)
WAIT FOR S_READY
;ENDFOLD

;FOLD PTP pt8 Vel=100 % PDAT82 Tool[1]:GUN_C1 Base[1]:ACTROS;%{PE}%R 8.2.20,%MKUKATPBASIS,%CMOVE,%VPTP,%P 1:PTP, 2:pt8, 3:, 5:100, 7:PDAT82
$BWDSTART=FALSE
PDAT_ACT=PPDAT82
FDAT_ACT=Fpt8
BAS(#PTP_PARAMS,100)
PTP Xpt8
;ENDFOLD
;FOLD PTP pt9 Vel=100 % PDAT83 Tool[1]:GUN_C1 Base[1]:ACTROS;%{PE}%R 8.2.20,%MKUKATPBASIS,%CMOVE,%VPTP,%P 1:PTP, 2:pt9, 3:, 5:100, 7:PDAT83
$BWDSTART=FALSE
PDAT_ACT=PPDAT83
FDAT_ACT=Fpt9
BAS(#PTP_PARAMS,100)
PTP Xpt9
;ENDFOLD
;FOLD PTP Xs_lx463 Vel=100 % P_OLP52 Tool[1]:GUN_C1 Base[1]:ACTROS;%{PE}%R 8.2.20,%MKUKATPBASIS,%CMOVE,%VPTP,%P 1:PTP, 2:Xs_lx463, 3:, 5:100, 7:P_OLP52
$BWDSTART=FALSE
PDAT_ACT=PP_OLP52
FDAT_ACT=FXs_lx463
BAS(#PTP_PARAMS,100)
PTP XXs_lx463
;ENDFOLD

;FOLD Collision.Monitoring_5_On ;%{PE}%MKUKATPUSER
COLLSTOP( 5, 1 ) ;not Interrupt-Controlled
;ENDFOLD
;FOLD Collision.Monitoring_AREA_6_Off . ;%{PE}%MKUKATPUSER
COLLSTOP( 12, 2+0 )
;ENDFOLD

;FOLD PTP Xs_lx464 CONT Vel=100 % P_OLP118 Tool[1]:GUN_C1 Base[1]:ACTROS;%{PE}%R 8.2.20,%MKUKATPBASIS,%CMOVE,%VPTP,%P 1:PTP, 2:Xs_lx464, 3:C_DIS, 5:100, 7:P_OLP118
$BWDSTART=FALSE
PDAT_ACT=PP_OLP118
FDAT_ACT=FXs_lx464
BAS(#PTP_PARAMS,100)
PTP XXs_lx464 C_DIS
;ENDFOLD

;FOLD ; swp_60_5096;%{PE}%R 8.2.20,%MKUKATPBASIS,%CCOMMENT,%VNORMAL,%P 2:swp_60_5096
;ENDFOLD
;FOLD PTP swp_60_5097 P_OLP119 SPOT Gun=1 RETR CLS PgNo1=32 ACTIVE=1 Tool[1]:GUN_C1 Base[1]:ACTROS;%{PE}%R 8.2.2,%MKUKATPSPOT,%CSPOT,%VPTP,%P 1:PTP, 2:swp_60_5097, 3:, 5:100, 7:P_OLP119, 10:1, 12:#FIRST, 14:#CLO, 16:32, 18:1, 20:1, 22:0, 24:1, 25:S_OLP19
$BWDSTART=FALSE
PDAT_ACT=PP_OLP119
FDAT_ACT=Fswp_60_5097
BAS(#PTP_PARAMS,PP_OLP119.VEL)
S_ACT.GUN=1
S_ACT.PAIR=SDEFAULT.PAIR
S_ACT.RETR=#CLO
S_ACT.CLO_TM=1
S_ACT.PGNO1=32
S_ACT.PGNO2=SDEFAULT.PGNO2
S_ACT.PRESS1=SDEFAULT.PRESS1
S_ACT.PRESS2=SDEFAULT.PRESS2
S_READY=FALSE
PTP Xswp_60_5097
USERSPOT(#SPOT, S_ACT)
WAIT FOR S_READY

;ENDFOLD

;FOLD ; swp_60_5098;%{PE}%R 8.2.20,%MKUKATPBASIS,%CCOMMENT,%VNORMAL,%P 2:swp_60_5098
;ENDFOLD
;FOLD PTP swp_60_5099 P_OLP120 SPOT Gun=1 RETR CLS PgNo1=31 ACTIVE=1 Tool[1]:GUN_C1 Base[1]:ACTROS;%{PE}%R 8.2.2,%MKUKATPSPOT,%CSPOT,%VPTP,%P 1:PTP, 2:swp_60_5099, 3:, 5:100, 7:P_OLP120, 10:1, 12:#FIRST, 14:#CLO, 16:31, 18:1, 20:1, 22:0, 24:1, 25:S_OLP18
$BWDSTART=FALSE
PDAT_ACT=PP_OLP120
FDAT_ACT=Fswp_60_5099
BAS(#PTP_PARAMS,PP_OLP120.VEL)
S_ACT.GUN=1
S_ACT.PAIR=SDEFAULT.PAIR
S_ACT.RETR=#CLO
S_ACT.CLO_TM=1
S_ACT.PGNO1=31
S_ACT.PGNO2=SDEFAULT.PGNO2
S_ACT.PRESS1=SDEFAULT.PRESS1
S_ACT.PRESS2=SDEFAULT.PRESS2
S_READY=FALSE
PTP Xswp_60_5099
USERSPOT(#SPOT, S_ACT)
WAIT FOR S_READY

;ENDFOLD

;FOLD ; swp_60_5100;%{PE}%R 8.2.20,%MKUKATPBASIS,%CCOMMENT,%VNORMAL,%P 2:swp_60_5100
;ENDFOLD
;FOLD PTP swp_60_5101 P_OLP121 SPOT Gun=1 RETR OPN PgNo1=30 ACTIVE=1 Tool[1]:GUN_C1 Base[1]:ACTROS;%{PE}%R 8.2.2,%MKUKATPSPOT,%CSPOT,%VPTP,%P 1:PTP, 2:swp_60_5101, 3:, 5:100, 7:P_OLP121, 10:1, 12:#FIRST, 14:#OPN, 16:30, 18:1, 20:1, 22:0, 24:1, 25:S_OLP17
$BWDSTART=FALSE
PDAT_ACT=PP_OLP121
FDAT_ACT=Fswp_60_5101
BAS(#PTP_PARAMS,PP_OLP121.VEL)
S_ACT.GUN=1
S_ACT.PAIR=SDEFAULT.PAIR
S_ACT.RETR=#OPN
S_ACT.CLO_TM=1
S_ACT.PGNO1=30
S_ACT.PGNO2=SDEFAULT.PGNO2
S_ACT.PRESS1=SDEFAULT.PRESS1
S_ACT.PRESS2=SDEFAULT.PRESS2
S_READY=FALSE
PTP Xswp_60_5101
USERSPOT(#SPOT, S_ACT)
WAIT FOR S_READY
;ENDFOLD

;FOLD PTP Xlx510 CONT Vel=100 % P_OLP59 Tool[1]:GUN_C1 Base[1]:ACTROS;%{PE}%R 8.2.20,%MKUKATPBASIS,%CMOVE,%VPTP,%P 1:PTP, 2:Xlx510, 3:C_DIS, 5:100, 7:P_OLP59
$BWDSTART=FALSE
PDAT_ACT=PP_OLP59
FDAT_ACT=FXlx510
BAS(#PTP_PARAMS,100)
PTP XXlx510 C_DIS
;ENDFOLD
;FOLD PTP Xlx511 CONT Vel=100 % P_OLP60 Tool[1]:GUN_C1 Base[1]:ACTROS;%{PE}%R 8.2.20,%MKUKATPBASIS,%CMOVE,%VPTP,%P 1:PTP, 2:Xlx511, 3:C_DIS, 5:100, 7:P_OLP60
$BWDSTART=FALSE
PDAT_ACT=PP_OLP60
FDAT_ACT=FXlx511
BAS(#PTP_PARAMS,100)
PTP XXlx511 C_DIS
;ENDFOLD

;FOLD ; swp_60_5084;%{PE}%R 8.2.20,%MKUKATPBASIS,%CCOMMENT,%VNORMAL,%P 2:swp_60_5084
;ENDFOLD
;FOLD PTP swp_60_5085 P_OLP122 SPOT Gun=1 RETR CLS PgNo1=35 ACTIVE=1 Tool[1]:GUN_C1 Base[1]:ACTROS;%{PE}%R 8.2.2,%MKUKATPSPOT,%CSPOT,%VPTP,%P 1:PTP, 2:swp_60_5085, 3:, 5:100, 7:P_OLP122, 10:1, 12:#FIRST, 14:#CLO, 16:35, 18:1, 20:1, 22:0, 24:1, 25:S_OLP22
$BWDSTART=FALSE
PDAT_ACT=PP_OLP122
FDAT_ACT=Fswp_60_5085
BAS(#PTP_PARAMS,PP_OLP122.VEL)
S_ACT.GUN=1
S_ACT.PAIR=SDEFAULT.PAIR
S_ACT.RETR=#CLO
S_ACT.CLO_TM=1
S_ACT.PGNO1=35
S_ACT.PGNO2=SDEFAULT.PGNO2
S_ACT.PRESS1=SDEFAULT.PRESS1
S_ACT.PRESS2=SDEFAULT.PRESS2
S_READY=FALSE
PTP Xswp_60_5085
USERSPOT(#SPOT, S_ACT)
WAIT FOR S_READY

;ENDFOLD

;FOLD PTP Xlx509 CONT Vel=100 % P_OLP61 Tool[1]:GUN_C1 Base[1]:ACTROS;%{PE}%R 8.2.20,%MKUKATPBASIS,%CMOVE,%VPTP,%P 1:PTP, 2:Xlx509, 3:C_DIS, 5:100, 7:P_OLP61
$BWDSTART=FALSE
PDAT_ACT=PP_OLP61
FDAT_ACT=FXlx509
BAS(#PTP_PARAMS,100)
PTP XXlx509 C_DIS
;ENDFOLD

;FOLD ; swp_60_5076;%{PE}%R 5.4.33,%MKUKATPBASIS,%CCOMMENT,%VNORMAL,%P 2:swp_60_5076
;ENDFOLD
;FOLD PTP swp_60_5076 P_OLP63 SPOT Gun=1 RETR OPN PgNo1=34 ACTIVE=1 Tool[1]:GUN_C1 Base[1]:ACTROS;%{PE}%R 8.2.2,%MKUKATPSPOT,%CSPOT,%VPTP,%P 1:PTP, 2:swp_60_5076, 3:, 5:100, 7:P_OLP63, 10:1, 12:#FIRST, 14:#OPN, 16:34, 18:1, 20:1, 22:0, 24:1, 25:S_OLP21
$BWDSTART=FALSE
PDAT_ACT=PP_OLP63
FDAT_ACT=Fswp_60_5076
BAS(#PTP_PARAMS,PP_OLP63.VEL)
S_ACT.GUN=1
S_ACT.PAIR=SDEFAULT.PAIR
S_ACT.RETR=#OPN
S_ACT.CLO_TM=1
S_ACT.PGNO1=34
S_ACT.PGNO2=SDEFAULT.PGNO2
S_ACT.PRESS1=SDEFAULT.PRESS1
S_ACT.PRESS2=SDEFAULT.PRESS2
S_READY=FALSE
PTP Xswp_60_5076
USERSPOT(#SPOT, S_ACT)
WAIT FOR S_READY
;ENDFOLD

;FOLD PTP pt11 CONT Vel=100 % PDAT85 Tool[1]:GUN_C1 Base[1]:ACTROS;%{PE}%R 8.2.20,%MKUKATPBASIS,%CMOVE,%VPTP,%P 1:PTP, 2:pt11, 3:C_DIS, 5:100, 7:PDAT85
$BWDSTART=FALSE
PDAT_ACT=PPDAT85
FDAT_ACT=Fpt11
BAS(#PTP_PARAMS,100)
PTP Xpt11 C_DIS
;ENDFOLD
;FOLD PTP pt12 CONT Vel=100 % PDAT86 Tool[1]:GUN_C1 Base[1]:ACTROS;%{PE}%R 8.2.20,%MKUKATPBASIS,%CMOVE,%VPTP,%P 1:PTP, 2:pt12, 3:C_DIS, 5:100, 7:PDAT86
$BWDSTART=FALSE
PDAT_ACT=PPDAT86
FDAT_ACT=Fpt12
BAS(#PTP_PARAMS,100)
PTP Xpt12 C_DIS
;ENDFOLD
;FOLD PTP pt13 CONT Vel=100 % PDAT87 Tool[1]:GUN_C1 Base[1]:ACTROS;%{PE}%R 8.2.20,%MKUKATPBASIS,%CMOVE,%VPTP,%P 1:PTP, 2:pt13, 3:C_DIS, 5:100, 7:PDAT87
$BWDSTART=FALSE
PDAT_ACT=PPDAT87
FDAT_ACT=Fpt13
BAS(#PTP_PARAMS,100)
PTP Xpt13 C_DIS
;ENDFOLD
;FOLD PTP pt14 Vel=100 % PDAT88 Tool[1]:GUN_C1 Base[1]:ACTROS;%{PE}%R 8.2.20,%MKUKATPBASIS,%CMOVE,%VPTP,%P 1:PTP, 2:pt14, 3:, 5:100, 7:PDAT88
$BWDSTART=FALSE
PDAT_ACT=PPDAT88
FDAT_ACT=Fpt14
BAS(#PTP_PARAMS,100)
PTP Xpt14
;ENDFOLD

;FOLD ; swp_60_5066;%{PE}%R 8.2.20,%MKUKATPBASIS,%CCOMMENT,%VNORMAL,%P 2:swp_60_5066
;ENDFOLD
;FOLD PTP swp_60_5066 PDAT89 SPOT Gun=1 RETR OPN PgNo1=48 ACTIVE=1 Tool[1]:GUN_C1 Base[1]:ACTROS;%{PE}%R 8.2.2,%MKUKATPSPOT,%CSPOT,%VPTP,%P 1:PTP, 2:swp_60_5066, 3:, 5:100, 7:PDAT89, 10:1, 12:#FIRST, 14:#OPN, 16:48, 18:1, 20:0, 22:0, 24:1, 25:NORMAL
$BWDSTART=FALSE
PDAT_ACT=PPDAT89
FDAT_ACT=Fswp_60_5066
BAS(#PTP_PARAMS,PPDAT89.VEL)
S_ACT.GUN=1
S_ACT.PAIR=SDEFAULT.PAIR
S_ACT.RETR=#OPN
S_ACT.CLO_TM=1
S_ACT.PGNO1=48
S_ACT.PGNO2=SDEFAULT.PGNO2
S_ACT.PRESS1=SDEFAULT.PRESS1
S_ACT.PRESS2=SDEFAULT.PRESS2
S_READY=FALSE
PTP Xswp_60_5066
USERSPOT(#SPOT, S_ACT)
WAIT FOR S_READY
;ENDFOLD

;FOLD PTP pt15 Vel=100 % PDAT90 Tool[1]:GUN_C1 Base[1]:ACTROS;%{PE}%R 8.2.20,%MKUKATPBASIS,%CMOVE,%VPTP,%P 1:PTP, 2:pt15, 3:, 5:100, 7:PDAT90
$BWDSTART=FALSE
PDAT_ACT=PPDAT90
FDAT_ACT=Fpt15
BAS(#PTP_PARAMS,100)
PTP Xpt15
;ENDFOLD
;FOLD PTP pt16 CONT Vel=100 % PDAT91 Tool[1]:GUN_C1 Base[1]:ACTROS;%{PE}%R 8.2.20,%MKUKATPBASIS,%CMOVE,%VPTP,%P 1:PTP, 2:pt16, 3:C_DIS, 5:100, 7:PDAT91
$BWDSTART=FALSE
PDAT_ACT=PPDAT91
FDAT_ACT=Fpt16
BAS(#PTP_PARAMS,100)
PTP Xpt16 C_DIS
;ENDFOLD
;FOLD PTP pt18 CONT Vel=100 % PDAT93 Tool[1]:GUN_C1 Base[1]:ACTROS;%{PE}%R 8.2.20,%MKUKATPBASIS,%CMOVE,%VPTP,%P 1:PTP, 2:pt18, 3:C_DIS, 5:100, 7:PDAT93
$BWDSTART=FALSE
PDAT_ACT=PPDAT93
FDAT_ACT=Fpt18
BAS(#PTP_PARAMS,100)
PTP Xpt18 C_DIS
;ENDFOLD
;FOLD PTP pt19 CONT Vel=100 % PDAT94 Tool[1]:GUN_C1 Base[1]:ACTROS;%{PE}%R 8.2.20,%MKUKATPBASIS,%CMOVE,%VPTP,%P 1:PTP, 2:pt19, 3:C_DIS, 5:100, 7:PDAT94
$BWDSTART=FALSE
PDAT_ACT=PPDAT94
FDAT_ACT=Fpt19
BAS(#PTP_PARAMS,100)
PTP Xpt19 C_DIS
;ENDFOLD

;FOLD PTP Xs_lx456 CONT Vel=100 % P_OLP64 Tool[1]:GUN_C1 Base[1]:ACTROS;%{PE}%R 8.2.20,%MKUKATPBASIS,%CMOVE,%VPTP,%P 1:PTP, 2:Xs_lx456, 3:C_DIS, 5:100, 7:P_OLP64
$BWDSTART=FALSE
PDAT_ACT=PP_OLP64
FDAT_ACT=FXs_lx456
BAS(#PTP_PARAMS,100)
PTP XXs_lx456 C_DIS
;ENDFOLD

;FOLD Collision.Monitoring_5_Off . ;%{PE}%MKUKATPUSER
COLLSTOP( 5, 2+0 )
;ENDFOLD

;FOLD PTP Xs_lx546 CONT Vel=100 % PDAT51 Tool[1]:GUN_C1 Base[1]:ACTROS;%{PE}%R 8.2.20,%MKUKATPBASIS,%CMOVE,%VPTP,%P 1:PTP, 2:Xs_lx546, 3:C_DIS, 5:100, 7:PDAT51
$BWDSTART=FALSE
PDAT_ACT=PPDAT51
FDAT_ACT=FXs_lx546
BAS(#PTP_PARAMS,100)
PTP XXs_lx546 C_DIS
;ENDFOLD
;FOLD PTP Xs_lx548 Vel=100 % PDAT53 Tool[1]:GUN_C1 Base[1]:ACTROS;%{PE}%R 8.2.20,%MKUKATPBASIS,%CMOVE,%VPTP,%P 1:PTP, 2:Xs_lx548, 3:, 5:100, 7:PDAT53
$BWDSTART=FALSE
PDAT_ACT=PPDAT53
FDAT_ACT=FXs_lx548
BAS(#PTP_PARAMS,100)
PTP XXs_lx548
;ENDFOLD
;FOLD PTP Xs_lx455 CONT Vel=100 % P_OLP69 Tool[1]:GUN_C1 Base[1]:ACTROS;%{PE}%R 8.2.19,%MKUKATPBASIS,%CMOVE,%VPTP,%P 1:PTP, 2:Xs_lx455, 3:C_DIS, 5:100, 7:P_OLP69
$BWDSTART=FALSE
PDAT_ACT=PP_OLP69
FDAT_ACT=FXs_lx455
BAS(#PTP_PARAMS,100)
PTP XXs_lx455 C_DIS
;ENDFOLD
;FOLD  ;%{PE}%R 8.2.20,%MKUKATPBASIS,%CCOMMENT,%VNORMAL,%P 2:
;ENDFOLD
;FOLD Collision.Monitoring_2_On ;%{PE}%MKUKATPUSER
COLLSTOP( 2, 1 ) ;Interrupt-Controlled
;ENDFOLD
;FOLD  ;%{PE}%R 8.2.20,%MKUKATPBASIS,%CCOMMENT,%VNORMAL,%P 2:
;ENDFOLD
;FOLD PTP pt20 CONT Vel=100 % PDAT95 Tool[1]:GUN_C1 Base[1]:ACTROS;%{PE}%R 8.2.20,%MKUKATPBASIS,%CMOVE,%VPTP,%P 1:PTP, 2:pt20, 3:C_DIS, 5:100, 7:PDAT95
$BWDSTART=FALSE
PDAT_ACT=PPDAT95
FDAT_ACT=Fpt20
BAS(#PTP_PARAMS,100)
PTP Xpt20 C_DIS
;ENDFOLD
;FOLD PTP P14 CONT Vel=100 % PDAT96 Tool[1]:GUN_C1 Base[1]:ACTROS;%{PE}%R 8.2.20,%MKUKATPBASIS,%CMOVE,%VPTP,%P 1:PTP, 2:P14, 3:C_DIS, 5:100, 7:PDAT96
$BWDSTART=FALSE
PDAT_ACT=PPDAT96
FDAT_ACT=FP14
BAS(#PTP_PARAMS,100)
PTP XP14 C_DIS
;ENDFOLD
;FOLD PTP Xs_lx449 CONT Vel=100 % P_OLP72 Tool[1]:GUN_C1 Base[1]:ACTROS;%{PE}%R 8.2.19,%MKUKATPBASIS,%CMOVE,%VPTP,%P 1:PTP, 2:Xs_lx449, 3:C_DIS, 5:100, 7:P_OLP72
$BWDSTART=FALSE
PDAT_ACT=PP_OLP72
FDAT_ACT=FXs_lx449
BAS(#PTP_PARAMS,100)
PTP XXs_lx449 C_DIS
;ENDFOLD

;FOLD ; swp_60_5626;%{PE}%R 5.4.33,%MKUKATPBASIS,%CCOMMENT,%VNORMAL,%P 2:swp_60_5626
;ENDFOLD
;FOLD PTP swp_60_5626 P_OLP73 SPOT Gun=1 RETR CLS PgNo1=36 ACTIVE=1 Tool[1]:GUN_C1 Base[1]:ACTROS;%{PE}%R 8.2.2,%MKUKATPSPOT,%CSPOT,%VPTP,%P 1:PTP, 2:swp_60_5626, 3:, 5:100, 7:P_OLP73, 10:1, 12:#FIRST, 14:#CLO, 16:36, 18:1, 20:1, 22:0, 24:1, 25:S_OLP23
$BWDSTART=FALSE
PDAT_ACT=PP_OLP73
FDAT_ACT=Fswp_60_5626
BAS(#PTP_PARAMS,PP_OLP73.VEL)
S_ACT.GUN=1
S_ACT.PAIR=SDEFAULT.PAIR
S_ACT.RETR=#CLO
S_ACT.CLO_TM=1
S_ACT.PGNO1=36
S_ACT.PGNO2=SDEFAULT.PGNO2
S_ACT.PRESS1=SDEFAULT.PRESS1
S_ACT.PRESS2=SDEFAULT.PRESS2
S_READY=FALSE
PTP Xswp_60_5626
USERSPOT(#SPOT, S_ACT)
WAIT FOR S_READY
;ENDFOLD

;FOLD ; swp_60_5640;%{PE}%R 5.4.33,%MKUKATPBASIS,%CCOMMENT,%VNORMAL,%P 2:swp_60_5640
;ENDFOLD
;FOLD PTP swp_60_5640 P_OLP74 SPOT Gun=1 RETR CLS PgNo1=37 ACTIVE=1 Tool[1]:GUN_C1 Base[1]:ACTROS;%{PE}%R 8.2.2,%MKUKATPSPOT,%CSPOT,%VPTP,%P 1:PTP, 2:swp_60_5640, 3:, 5:100, 7:P_OLP74, 10:1, 12:#FIRST, 14:#CLO, 16:37, 18:1, 20:1, 22:0, 24:1, 25:S_OLP24
$BWDSTART=FALSE
PDAT_ACT=PP_OLP74
FDAT_ACT=Fswp_60_5640
BAS(#PTP_PARAMS,PP_OLP74.VEL)
S_ACT.GUN=1
S_ACT.PAIR=SDEFAULT.PAIR
S_ACT.RETR=#CLO
S_ACT.CLO_TM=1
S_ACT.PGNO1=37
S_ACT.PGNO2=SDEFAULT.PGNO2
S_ACT.PRESS1=SDEFAULT.PRESS1
S_ACT.PRESS2=SDEFAULT.PRESS2
S_READY=FALSE
PTP Xswp_60_5640
USERSPOT(#SPOT, S_ACT)
WAIT FOR S_READY
;ENDFOLD

;FOLD PTP Xs_lx447 CONT Vel=100 % P_OLP75 Tool[1]:GUN_C1 Base[1]:ACTROS;%{PE}%R 8.2.19,%MKUKATPBASIS,%CMOVE,%VPTP,%P 1:PTP, 2:Xs_lx447, 3:C_DIS, 5:100, 7:P_OLP75
$BWDSTART=FALSE
PDAT_ACT=PP_OLP75
FDAT_ACT=FXs_lx447
BAS(#PTP_PARAMS,100)
PTP XXs_lx447 C_DIS
;ENDFOLD
;FOLD PTP Xs_lx448 CONT Vel=100 % P_OLP76 Tool[1]:GUN_C1 Base[1]:ACTROS;%{PE}%R 8.2.19,%MKUKATPBASIS,%CMOVE,%VPTP,%P 1:PTP, 2:Xs_lx448, 3:C_DIS, 5:100, 7:P_OLP76
$BWDSTART=FALSE
PDAT_ACT=PP_OLP76
FDAT_ACT=FXs_lx448
BAS(#PTP_PARAMS,100)
PTP XXs_lx448 C_DIS
;ENDFOLD
;FOLD PTP P15 CONT Vel=100 % PDAT97 Tool[1]:GUN_C1 Base[1]:ACTROS;%{PE}%R 8.2.20,%MKUKATPBASIS,%CMOVE,%VPTP,%P 1:PTP, 2:P15, 3:C_DIS, 5:100, 7:PDAT97
$BWDSTART=FALSE
PDAT_ACT=PPDAT97
FDAT_ACT=FP15
BAS(#PTP_PARAMS,100)
PTP XP15 C_DIS
;ENDFOLD

;FOLD PTP Xs_lx446 CONT Vel=100 % P_OLP77 Tool[1]:GUN_C1 Base[1]:ACTROS;%{PE}%R 8.2.20,%MKUKATPBASIS,%CMOVE,%VPTP,%P 1:PTP, 2:Xs_lx446, 3:C_DIS, 5:100, 7:P_OLP77
$BWDSTART=FALSE
PDAT_ACT=PP_OLP77
FDAT_ACT=FXs_lx446
BAS(#PTP_PARAMS,100)
PTP XXs_lx446 C_DIS
;ENDFOLD
;FOLD PTP Xs_lx445 CONT Vel=100 % P_OLP78 Tool[1]:GUN_C1 Base[1]:ACTROS;%{PE}%R 8.2.20,%MKUKATPBASIS,%CMOVE,%VPTP,%P 1:PTP, 2:Xs_lx445, 3:C_DIS, 5:100, 7:P_OLP78
$BWDSTART=FALSE
PDAT_ACT=PP_OLP78
FDAT_ACT=FXs_lx445
BAS(#PTP_PARAMS,100)
PTP XXs_lx445 C_DIS
;ENDFOLD

;FOLD ; swp_60_5060;%{PE}%R 5.4.33,%MKUKATPBASIS,%CCOMMENT,%VNORMAL,%P 2:swp_60_5060
;ENDFOLD
;FOLD PTP swp_60_5060 P_OLP79 SPOT Gun=1 RETR CLS PgNo1=38 ACTIVE=1 Tool[1]:GUN_C1 Base[1]:ACTROS;%{PE}%R 8.2.2,%MKUKATPSPOT,%CSPOT,%VPTP,%P 1:PTP, 2:swp_60_5060, 3:, 5:100, 7:P_OLP79, 10:1, 12:#FIRST, 14:#CLO, 16:38, 18:1, 20:1, 22:0, 24:1, 25:S_OLP25
$BWDSTART=FALSE
PDAT_ACT=PP_OLP79
FDAT_ACT=Fswp_60_5060
BAS(#PTP_PARAMS,PP_OLP79.VEL)
S_ACT.GUN=1
S_ACT.PAIR=SDEFAULT.PAIR
S_ACT.RETR=#CLO
S_ACT.CLO_TM=1
S_ACT.PGNO1=38
S_ACT.PGNO2=SDEFAULT.PGNO2
S_ACT.PRESS1=SDEFAULT.PRESS1
S_ACT.PRESS2=SDEFAULT.PRESS2
S_READY=FALSE
PTP Xswp_60_5060
USERSPOT(#SPOT, S_ACT)
WAIT FOR S_READY
;ENDFOLD

;FOLD PTP Xs_lx442 CONT Vel=100 % P_OLP80 Tool[1]:GUN_C1 Base[1]:ACTROS;%{PE}%R 8.2.20,%MKUKATPBASIS,%CMOVE,%VPTP,%P 1:PTP, 2:Xs_lx442, 3:C_DIS, 5:100, 7:P_OLP80
$BWDSTART=FALSE
PDAT_ACT=PP_OLP80
FDAT_ACT=FXs_lx442
BAS(#PTP_PARAMS,100)
PTP XXs_lx442 C_DIS
;ENDFOLD
;FOLD PTP Xs_lx444 CONT Vel=100 % P_OLP81 Tool[1]:GUN_C1 Base[1]:ACTROS;%{PE}%R 8.2.20,%MKUKATPBASIS,%CMOVE,%VPTP,%P 1:PTP, 2:Xs_lx444, 3:C_DIS, 5:100, 7:P_OLP81
$BWDSTART=FALSE
PDAT_ACT=PP_OLP81
FDAT_ACT=FXs_lx444
BAS(#PTP_PARAMS,100)
PTP XXs_lx444 C_DIS
;ENDFOLD

;FOLD PTP Xs_lx443 CONT Vel=100 % P_OLP82 Tool[1]:GUN_C1 Base[1]:ACTROS;%{PE}%R 8.2.20,%MKUKATPBASIS,%CMOVE,%VPTP,%P 1:PTP, 2:Xs_lx443, 3:C_DIS, 5:100, 7:P_OLP82
$BWDSTART=FALSE
PDAT_ACT=PP_OLP82
FDAT_ACT=FXs_lx443
BAS(#PTP_PARAMS,100)
PTP XXs_lx443 C_DIS
;ENDFOLD
;FOLD PTP Xs_lx520 CONT Vel=100 % PDAT24 Tool[1]:GUN_C1 Base[1]:ACTROS;%{PE}%R 8.2.20,%MKUKATPBASIS,%CMOVE,%VPTP,%P 1:PTP, 2:Xs_lx520, 3:C_DIS, 5:100, 7:PDAT24
$BWDSTART=FALSE
PDAT_ACT=PPDAT24
FDAT_ACT=FXs_lx520
BAS(#PTP_PARAMS,100)
PTP XXs_lx520 C_DIS
;ENDFOLD

;FOLD ; swp_60_5056;%{PE}%R 5.4.33,%MKUKATPBASIS,%CCOMMENT,%VNORMAL,%P 2:swp_60_5056
;ENDFOLD
;FOLD PTP swp_60_5056 P_OLP85 SPOT Gun=1 RETR CLS PgNo1=39 ACTIVE=1 Tool[1]:GUN_C1 Base[1]:ACTROS;%{PE}%R 8.2.2,%MKUKATPSPOT,%CSPOT,%VPTP,%P 1:PTP, 2:swp_60_5056, 3:, 5:100, 7:P_OLP85, 10:1, 12:#FIRST, 14:#CLO, 16:39, 18:1, 20:1, 22:0, 24:1, 25:S_OLP26
$BWDSTART=FALSE
PDAT_ACT=PP_OLP85
FDAT_ACT=Fswp_60_5056
BAS(#PTP_PARAMS,PP_OLP85.VEL)
S_ACT.GUN=1
S_ACT.PAIR=SDEFAULT.PAIR
S_ACT.RETR=#CLO
S_ACT.CLO_TM=1
S_ACT.PGNO1=39
S_ACT.PGNO2=SDEFAULT.PGNO2
S_ACT.PRESS1=SDEFAULT.PRESS1
S_ACT.PRESS2=SDEFAULT.PRESS2
S_READY=FALSE
PTP Xswp_60_5056
USERSPOT(#SPOT, S_ACT)
WAIT FOR S_READY
;ENDFOLD

;FOLD PTP Xs_lx521 CONT Vel=100 % PDAT25 Tool[1]:GUN_C1 Base[1]:ACTROS;%{PE}%R 8.2.20,%MKUKATPBASIS,%CMOVE,%VPTP,%P 1:PTP, 2:Xs_lx521, 3:C_DIS, 5:100, 7:PDAT25
$BWDSTART=FALSE
PDAT_ACT=PPDAT25
FDAT_ACT=FXs_lx521
BAS(#PTP_PARAMS,100)
PTP XXs_lx521 C_DIS
;ENDFOLD

;FOLD ; swp_60_5058;%{PE}%R 5.4.33,%MKUKATPBASIS,%CCOMMENT,%VNORMAL,%P 2:swp_60_5058
;ENDFOLD
;FOLD PTP swp_60_5058 P_OLP86 SPOT Gun=1 RETR CLS PgNo1=40 ACTIVE=1 Tool[1]:GUN_C1 Base[1]:ACTROS;%{PE}%R 8.2.2,%MKUKATPSPOT,%CSPOT,%VPTP,%P 1:PTP, 2:swp_60_5058, 3:, 5:100, 7:P_OLP86, 10:1, 12:#FIRST, 14:#CLO, 16:40, 18:1, 20:1, 22:0, 24:1, 25:S_OLP27
$BWDSTART=FALSE
PDAT_ACT=PP_OLP86
FDAT_ACT=Fswp_60_5058
BAS(#PTP_PARAMS,PP_OLP86.VEL)
S_ACT.GUN=1
S_ACT.PAIR=SDEFAULT.PAIR
S_ACT.RETR=#CLO
S_ACT.CLO_TM=1
S_ACT.PGNO1=40
S_ACT.PGNO2=SDEFAULT.PGNO2
S_ACT.PRESS1=SDEFAULT.PRESS1
S_ACT.PRESS2=SDEFAULT.PRESS2
S_READY=FALSE
PTP Xswp_60_5058
USERSPOT(#SPOT, S_ACT)
WAIT FOR S_READY
;ENDFOLD

;FOLD PTP Xs_lx522 CONT Vel=100 % PDAT26 Tool[1]:GUN_C1 Base[1]:ACTROS;%{PE}%R 8.2.20,%MKUKATPBASIS,%CMOVE,%VPTP,%P 1:PTP, 2:Xs_lx522, 3:C_DIS, 5:100, 7:PDAT26
$BWDSTART=FALSE
PDAT_ACT=PPDAT26
FDAT_ACT=FXs_lx522
BAS(#PTP_PARAMS,100)
PTP XXs_lx522 C_DIS
;ENDFOLD
;FOLD PTP Xs_lx437 CONT Vel=100 % P_OLP88 Tool[1]:GUN_C1 Base[1]:ACTROS;%{PE}%R 8.2.20,%MKUKATPBASIS,%CMOVE,%VPTP,%P 1:PTP, 2:Xs_lx437, 3:C_DIS, 5:100, 7:P_OLP88
$BWDSTART=FALSE
PDAT_ACT=PP_OLP88
FDAT_ACT=FXs_lx437
BAS(#PTP_PARAMS,100)
PTP XXs_lx437 C_DIS
;ENDFOLD
;FOLD PTP Xs_lx439 CONT Vel=100 % P_OLP89 Tool[1]:GUN_C1 Base[1]:ACTROS;%{PE}%R 8.2.20,%MKUKATPBASIS,%CMOVE,%VPTP,%P 1:PTP, 2:Xs_lx439, 3:C_DIS, 5:100, 7:P_OLP89
$BWDSTART=FALSE
PDAT_ACT=PP_OLP89
FDAT_ACT=FXs_lx439
BAS(#PTP_PARAMS,100)
PTP XXs_lx439 C_DIS
;ENDFOLD
;FOLD PTP Xs_lx524 CONT Vel=100 % PDAT28 Tool[1]:GUN_C1 Base[1]:ACTROS;%{PE}%R 8.2.20,%MKUKATPBASIS,%CMOVE,%VPTP,%P 1:PTP, 2:Xs_lx524, 3:C_DIS, 5:100, 7:PDAT28
$BWDSTART=FALSE
PDAT_ACT=PPDAT28
FDAT_ACT=FXs_lx524
BAS(#PTP_PARAMS,100)
PTP XXs_lx524 C_DIS
;ENDFOLD

;FOLD ; swp_60_5424;%{PE}%R 5.4.33,%MKUKATPBASIS,%CCOMMENT,%VNORMAL,%P 2:swp_60_5424
;ENDFOLD
;FOLD PTP swp_60_5424 P_OLP91 SPOT Gun=1 RETR OPN PgNo1=41 ACTIVE=1 Tool[1]:GUN_C1 Base[1]:ACTROS;%{PE}%R 8.2.2,%MKUKATPSPOT,%CSPOT,%VPTP,%P 1:PTP, 2:swp_60_5424, 3:, 5:100, 7:P_OLP91, 10:1, 12:#FIRST, 14:#OPN, 16:41, 18:1, 20:1, 22:0, 24:1, 25:S_OLP28
$BWDSTART=FALSE
PDAT_ACT=PP_OLP91
FDAT_ACT=Fswp_60_5424
BAS(#PTP_PARAMS,PP_OLP91.VEL)
S_ACT.GUN=1
S_ACT.PAIR=SDEFAULT.PAIR
S_ACT.RETR=#OPN
S_ACT.CLO_TM=1
S_ACT.PGNO1=41
S_ACT.PGNO2=SDEFAULT.PGNO2
S_ACT.PRESS1=SDEFAULT.PRESS1
S_ACT.PRESS2=SDEFAULT.PRESS2
S_READY=FALSE
PTP Xswp_60_5424
USERSPOT(#SPOT, S_ACT)
WAIT FOR S_READY
;ENDFOLD

;FOLD PTP Xs_lx434 CONT Vel=100 % P_OLP92 Tool[1]:GUN_C1 Base[1]:ACTROS;%{PE}%R 8.2.20,%MKUKATPBASIS,%CMOVE,%VPTP,%P 1:PTP, 2:Xs_lx434, 3:C_DIS, 5:100, 7:P_OLP92
$BWDSTART=FALSE
PDAT_ACT=PP_OLP92
FDAT_ACT=FXs_lx434
BAS(#PTP_PARAMS,100)
PTP XXs_lx434 C_DIS
;ENDFOLD
;FOLD PTP Xs_lx435 CONT Vel=100 % P_OLP93 Tool[1]:GUN_C1 Base[1]:ACTROS;%{PE}%R 8.2.20,%MKUKATPBASIS,%CMOVE,%VPTP,%P 1:PTP, 2:Xs_lx435, 3:C_DIS, 5:100, 7:P_OLP93
$BWDSTART=FALSE
PDAT_ACT=PP_OLP93
FDAT_ACT=FXs_lx435
BAS(#PTP_PARAMS,100)
PTP XXs_lx435 C_DIS
;ENDFOLD
;FOLD PTP Xs_lx525 CONT Vel=100 % PDAT29 Tool[1]:GUN_C1 Base[1]:ACTROS;%{PE}%R 8.2.20,%MKUKATPBASIS,%CMOVE,%VPTP,%P 1:PTP, 2:Xs_lx525, 3:C_DIS, 5:100, 7:PDAT29
$BWDSTART=FALSE
PDAT_ACT=PPDAT29
FDAT_ACT=FXs_lx525
BAS(#PTP_PARAMS,100)
PTP XXs_lx525 C_DIS
;ENDFOLD
;FOLD PTP Xs_lx527 CONT Vel=100 % PDAT31 Tool[1]:GUN_C1 Base[1]:ACTROS;%{PE}%R 8.2.20,%MKUKATPBASIS,%CMOVE,%VPTP,%P 1:PTP, 2:Xs_lx527, 3:C_DIS, 5:100, 7:PDAT31
$BWDSTART=FALSE
PDAT_ACT=PPDAT31
FDAT_ACT=FXs_lx527
BAS(#PTP_PARAMS,100)
PTP XXs_lx527 C_DIS
;ENDFOLD
;FOLD PTP Xs_lx526 CONT Vel=100 % PDAT30 Tool[1]:GUN_C1 Base[1]:ACTROS;%{PE}%R 8.2.20,%MKUKATPBASIS,%CMOVE,%VPTP,%P 1:PTP, 2:Xs_lx526, 3:C_DIS, 5:100, 7:PDAT30
$BWDSTART=FALSE
PDAT_ACT=PPDAT30
FDAT_ACT=FXs_lx526
BAS(#PTP_PARAMS,100)
PTP XXs_lx526 C_DIS
;ENDFOLD
;FOLD PTP Xs_lx431 CONT Vel=100 % P_OLP96 Tool[1]:GUN_C1 Base[1]:ACTROS;%{PE}%R 8.2.20,%MKUKATPBASIS,%CMOVE,%VPTP,%P 1:PTP, 2:Xs_lx431, 3:C_DIS, 5:100, 7:P_OLP96
$BWDSTART=FALSE
PDAT_ACT=PP_OLP96
FDAT_ACT=FXs_lx431
BAS(#PTP_PARAMS,100)
PTP XXs_lx431 C_DIS
;ENDFOLD
;FOLD PTP Xs_lx430 CONT Vel=100 % P_OLP97 Tool[1]:GUN_C1 Base[1]:ACTROS;%{PE}%R 8.2.20,%MKUKATPBASIS,%CMOVE,%VPTP,%P 1:PTP, 2:Xs_lx430, 3:C_DIS, 5:100, 7:P_OLP97
$BWDSTART=FALSE
PDAT_ACT=PP_OLP97
FDAT_ACT=FXs_lx430
BAS(#PTP_PARAMS,100)
PTP XXs_lx430 C_DIS
;ENDFOLD

;FOLD ; swp_60_5430;%{PE}%R 5.4.33,%MKUKATPBASIS,%CCOMMENT,%VNORMAL,%P 2:swp_60_5430
;ENDFOLD
;FOLD PTP swp_60_5430 P_OLP100 SPOT Gun=1 RETR CLS PgNo1=42 ACTIVE=1 Tool[1]:GUN_C1 Base[1]:ACTROS;%{PE}%R 8.2.2,%MKUKATPSPOT,%CSPOT,%VPTP,%P 1:PTP, 2:swp_60_5430, 3:, 5:100, 7:P_OLP100, 10:1, 12:#FIRST, 14:#CLO, 16:42, 18:1, 20:1, 22:0, 24:1, 25:S_OLP29
$BWDSTART=FALSE
PDAT_ACT=PP_OLP100
FDAT_ACT=Fswp_60_5430
BAS(#PTP_PARAMS,PP_OLP100.VEL)
S_ACT.GUN=1
S_ACT.PAIR=SDEFAULT.PAIR
S_ACT.RETR=#CLO
S_ACT.CLO_TM=1
S_ACT.PGNO1=42
S_ACT.PGNO2=SDEFAULT.PGNO2
S_ACT.PRESS1=SDEFAULT.PRESS1
S_ACT.PRESS2=SDEFAULT.PRESS2
S_READY=FALSE
PTP Xswp_60_5430
USERSPOT(#SPOT, S_ACT)
WAIT FOR S_READY
;ENDFOLD

;FOLD ; swp_60_5432;%{PE}%R 5.4.33,%MKUKATPBASIS,%CCOMMENT,%VNORMAL,%P 2:swp_60_5432
;ENDFOLD
;FOLD PTP swp_60_5432 P_OLP101 SPOT Gun=1 RETR CLS PgNo1=43 ACTIVE=1 Tool[1]:GUN_C1 Base[1]:ACTROS;%{PE}%R 8.2.2,%MKUKATPSPOT,%CSPOT,%VPTP,%P 1:PTP, 2:swp_60_5432, 3:, 5:100, 7:P_OLP101, 10:1, 12:#FIRST, 14:#CLO, 16:43, 18:1, 20:1, 22:0, 24:1, 25:S_OLP30
$BWDSTART=FALSE
PDAT_ACT=PP_OLP101
FDAT_ACT=Fswp_60_5432
BAS(#PTP_PARAMS,PP_OLP101.VEL)
S_ACT.GUN=1
S_ACT.PAIR=SDEFAULT.PAIR
S_ACT.RETR=#CLO
S_ACT.CLO_TM=1
S_ACT.PGNO1=43
S_ACT.PGNO2=SDEFAULT.PGNO2
S_ACT.PRESS1=SDEFAULT.PRESS1
S_ACT.PRESS2=SDEFAULT.PRESS2
S_READY=FALSE
PTP Xswp_60_5432
USERSPOT(#SPOT, S_ACT)
WAIT FOR S_READY
;ENDFOLD

;FOLD ; swp_60_5434;%{PE}%R 5.4.33,%MKUKATPBASIS,%CCOMMENT,%VNORMAL,%P 2:swp_60_5434
;ENDFOLD
;FOLD PTP swp_60_5434 P_OLP102 SPOT Gun=1 RETR CLS PgNo1=44 ACTIVE=1 Tool[1]:GUN_C1 Base[1]:ACTROS;%{PE}%R 8.2.2,%MKUKATPSPOT,%CSPOT,%VPTP,%P 1:PTP, 2:swp_60_5434, 3:, 5:100, 7:P_OLP102, 10:1, 12:#FIRST, 14:#CLO, 16:44, 18:1, 20:1, 22:0, 24:1, 25:S_OLP31
$BWDSTART=FALSE
PDAT_ACT=PP_OLP102
FDAT_ACT=Fswp_60_5434
BAS(#PTP_PARAMS,PP_OLP102.VEL)
S_ACT.GUN=1
S_ACT.PAIR=SDEFAULT.PAIR
S_ACT.RETR=#CLO
S_ACT.CLO_TM=1
S_ACT.PGNO1=44
S_ACT.PGNO2=SDEFAULT.PGNO2
S_ACT.PRESS1=SDEFAULT.PRESS1
S_ACT.PRESS2=SDEFAULT.PRESS2
S_READY=FALSE
PTP Xswp_60_5434
USERSPOT(#SPOT, S_ACT)
WAIT FOR S_READY
;ENDFOLD

;FOLD PTP Xs_lx531 CONT Vel=100 % PDAT35 Tool[1]:GUN_C1 Base[1]:ACTROS;%{PE}%R 8.2.20,%MKUKATPBASIS,%CMOVE,%VPTP,%P 1:PTP, 2:Xs_lx531, 3:C_DIS, 5:100, 7:PDAT35
$BWDSTART=FALSE
PDAT_ACT=PPDAT35
FDAT_ACT=FXs_lx531
BAS(#PTP_PARAMS,100)
PTP XXs_lx531 C_DIS
;ENDFOLD
;FOLD PTP Xs_lx532 CONT Vel=100 % PDAT36 Tool[1]:GUN_C1 Base[1]:ACTROS;%{PE}%R 8.2.20,%MKUKATPBASIS,%CMOVE,%VPTP,%P 1:PTP, 2:Xs_lx532, 3:C_DIS, 5:100, 7:PDAT36
$BWDSTART=FALSE
PDAT_ACT=PPDAT36
FDAT_ACT=FXs_lx532
BAS(#PTP_PARAMS,100)
PTP XXs_lx532 C_DIS
;ENDFOLD

;FOLD ; swp_60_5436;%{PE}%R 5.4.33,%MKUKATPBASIS,%CCOMMENT,%VNORMAL,%P 2:swp_60_5436
;ENDFOLD
;FOLD PTP swp_60_5436 P_OLP105 SPOT Gun=1 RETR CLS PgNo1=45 ACTIVE=1 Tool[1]:GUN_C1 Base[1]:ACTROS;%{PE}%R 8.2.2,%MKUKATPSPOT,%CSPOT,%VPTP,%P 1:PTP, 2:swp_60_5436, 3:, 5:100, 7:P_OLP105, 10:1, 12:#FIRST, 14:#CLO, 16:45, 18:1, 20:1, 22:0, 24:1, 25:S_OLP32
$BWDSTART=FALSE
PDAT_ACT=PP_OLP105
FDAT_ACT=Fswp_60_5436
BAS(#PTP_PARAMS,PP_OLP105.VEL)
S_ACT.GUN=1
S_ACT.PAIR=SDEFAULT.PAIR
S_ACT.RETR=#CLO
S_ACT.CLO_TM=1
S_ACT.PGNO1=45
S_ACT.PGNO2=SDEFAULT.PGNO2
S_ACT.PRESS1=SDEFAULT.PRESS1
S_ACT.PRESS2=SDEFAULT.PRESS2
S_READY=FALSE
PTP Xswp_60_5436
USERSPOT(#SPOT, S_ACT)
WAIT FOR S_READY
;ENDFOLD

;FOLD ; swp_60_5438;%{PE}%R 5.4.33,%MKUKATPBASIS,%CCOMMENT,%VNORMAL,%P 2:swp_60_5438
;ENDFOLD
;FOLD PTP swp_60_5438 P_OLP107 SPOT Gun=1 RETR CLS PgNo1=46 ACTIVE=1 Tool[1]:GUN_C1 Base[1]:ACTROS;%{PE}%R 8.2.2,%MKUKATPSPOT,%CSPOT,%VPTP,%P 1:PTP, 2:swp_60_5438, 3:, 5:100, 7:P_OLP107, 10:1, 12:#FIRST, 14:#CLO, 16:46, 18:1, 20:1, 22:0, 24:1, 25:S_OLP33
$BWDSTART=FALSE
PDAT_ACT=PP_OLP107
FDAT_ACT=Fswp_60_5438
BAS(#PTP_PARAMS,PP_OLP107.VEL)
S_ACT.GUN=1
S_ACT.PAIR=SDEFAULT.PAIR
S_ACT.RETR=#CLO
S_ACT.CLO_TM=1
S_ACT.PGNO1=46
S_ACT.PGNO2=SDEFAULT.PGNO2
S_ACT.PRESS1=SDEFAULT.PRESS1
S_ACT.PRESS2=SDEFAULT.PRESS2
S_READY=FALSE
PTP Xswp_60_5438
USERSPOT(#SPOT, S_ACT)
WAIT FOR S_READY
;ENDFOLD

;FOLD ; swp_60_5440;%{PE}%R 5.4.33,%MKUKATPBASIS,%CCOMMENT,%VNORMAL,%P 2:swp_60_5440
;ENDFOLD
;FOLD PTP swp_60_5440 P_OLP108 SPOT Gun=1 RETR CLS PgNo1=47 ACTIVE=1 Tool[1]:GUN_C1 Base[1]:ACTROS;%{PE}%R 8.2.2,%MKUKATPSPOT,%CSPOT,%VPTP,%P 1:PTP, 2:swp_60_5440, 3:, 5:100, 7:P_OLP108, 10:1, 12:#FIRST, 14:#CLO, 16:47, 18:1, 20:1, 22:0, 24:1, 25:S_OLP34
$BWDSTART=FALSE
PDAT_ACT=PP_OLP108
FDAT_ACT=Fswp_60_5440
BAS(#PTP_PARAMS,PP_OLP108.VEL)
S_ACT.GUN=1
S_ACT.PAIR=SDEFAULT.PAIR
S_ACT.RETR=#CLO
S_ACT.CLO_TM=1
S_ACT.PGNO1=47
S_ACT.PGNO2=SDEFAULT.PGNO2
S_ACT.PRESS1=SDEFAULT.PRESS1
S_ACT.PRESS2=SDEFAULT.PRESS2
S_READY=FALSE
PTP Xswp_60_5440
USERSPOT(#SPOT, S_ACT)
WAIT FOR S_READY
;ENDFOLD

;FOLD PTP Xs_lx421 CONT Vel=100 % P_OLP109 Tool[1]:GUN_C1 Base[1]:ACTROS;%{PE}%R 8.2.20,%MKUKATPBASIS,%CMOVE,%VPTP,%P 1:PTP, 2:Xs_lx421, 3:C_DIS, 5:100, 7:P_OLP109
$BWDSTART=FALSE
PDAT_ACT=PP_OLP109
FDAT_ACT=FXs_lx421
BAS(#PTP_PARAMS,100)
PTP XXs_lx421 C_DIS
;ENDFOLD
;FOLD PTP Xs_lx422 CONT Vel=100 % P_OLP110 Tool[1]:GUN_C1 Base[1]:ACTROS;%{PE}%R 8.2.20,%MKUKATPBASIS,%CMOVE,%VPTP,%P 1:PTP, 2:Xs_lx422, 3:C_DIS, 5:100, 7:P_OLP110
$BWDSTART=FALSE
PDAT_ACT=PP_OLP110
FDAT_ACT=FXs_lx422
BAS(#PTP_PARAMS,100)
PTP XXs_lx422 C_DIS
;ENDFOLD
;FOLD PTP Xs_lx534 CONT Vel=100 % PDAT38 Tool[1]:GUN_C1 Base[1]:ACTROS;%{PE}%R 8.2.20,%MKUKATPBASIS,%CMOVE,%VPTP,%P 1:PTP, 2:Xs_lx534, 3:C_DIS, 5:100, 7:PDAT38
$BWDSTART=FALSE
PDAT_ACT=PPDAT38
FDAT_ACT=FXs_lx534
BAS(#PTP_PARAMS,100)
PTP XXs_lx534 C_DIS
;ENDFOLD
;FOLD PTP Xs_lx423 CONT Vel=100 % P_OLP111 Tool[1]:GUN_C1 Base[1]:ACTROS;%{PE}%R 8.2.20,%MKUKATPBASIS,%CMOVE,%VPTP,%P 1:PTP, 2:Xs_lx423, 3:C_DIS, 5:100, 7:P_OLP111
$BWDSTART=FALSE
PDAT_ACT=PP_OLP111
FDAT_ACT=FXs_lx423
BAS(#PTP_PARAMS,100)
PTP XXs_lx423 C_DIS
;ENDFOLD
;FOLD PTP Xs_lx424 CONT Vel=100 % P_OLP112 Tool[1]:GUN_C1 Base[1]:ACTROS;%{PE}%R 8.2.20,%MKUKATPBASIS,%CMOVE,%VPTP,%P 1:PTP, 2:Xs_lx424, 3:C_DIS, 5:100, 7:P_OLP112
$BWDSTART=FALSE
PDAT_ACT=PP_OLP112
FDAT_ACT=FXs_lx424
BAS(#PTP_PARAMS,100)
PTP XXs_lx424 C_DIS
;ENDFOLD

;FOLD OUT 3348 'Fora area GEOBOX' State=TRUE ;%{PE}%R 8.2.20,%MKUKATPBASIS,%COUT,%VOUTX,%P 2:3348, 3:Fora area GEOBOX, 5:TRUE, 6:
$OUT[3348]=TRUE
;ENDFOLD
end_weld_GEO()              ; Bit fim solda GEO

;FOLD PTP Xs_lx535 CONT Vel=100 % PDAT39 Tool[1]:GUN_C1 Base[1]:ACTROS;%{PE}%R 8.2.20,%MKUKATPBASIS,%CMOVE,%VPTP,%P 1:PTP, 2:Xs_lx535, 3:C_DIS, 5:100, 7:PDAT39
$BWDSTART=FALSE
PDAT_ACT=PPDAT39
FDAT_ACT=FXs_lx535
BAS(#PTP_PARAMS,100)
PTP XXs_lx535 C_DIS
;ENDFOLD
;FOLD PTP Xs_lx537 Vel=100 % PDAT41 Tool[1]:GUN_C1 Base[1]:ACTROS;%{PE}%R 8.2.20,%MKUKATPBASIS,%CMOVE,%VPTP,%P 1:PTP, 2:Xs_lx537, 3:, 5:100, 7:PDAT41
$BWDSTART=FALSE
PDAT_ACT=PPDAT41
FDAT_ACT=FXs_lx537
BAS(#PTP_PARAMS,100)
PTP XXs_lx537
;ENDFOLD

;FOLD Collision.Monitoring_2_Off . ;%{PE}%MKUKATPUSER
COLLSTOP( 2, 2+0 )
;ENDFOLD

;FOLD PTP Xs_lx386 CONT Vel=100 % P_OLP113 Tool[1]:GUN_C1 Base[1]:ACTROS;%{PE}%R 8.2.20,%MKUKATPBASIS,%CMOVE,%VPTP,%P 1:PTP, 2:Xs_lx386, 3:C_DIS, 5:100, 7:P_OLP113
$BWDSTART=FALSE
PDAT_ACT=PP_OLP113
FDAT_ACT=FXs_lx386
BAS(#PTP_PARAMS,100)
PTP XXs_lx386 C_DIS
;ENDFOLD

IF (NOT(GHOST())) THEN
if FraesAnf (1) then
  f_fraes1 ()
endif
ENDIF

END

--- ps_com_geo_c1.dat ---
&ACCESS RVO1
&REL 24
&COMMENT Solda GUN C1 Geometria
&PARAM DISKPATH = KRC:\R1\Program\SOLDA LTC
DEFDAT  ps_com_geo_c1
;FOLD EXTERNAL DECLARATIONS;%{PE}%MKUKATPBASIS,%CEXT,%VCOMMON,%P
;FOLD GRIPPERTECH EXT
EXT  H50 (INT  :IN,INT  :IN,INT  :IN,GRP_TYP  :IN )
;ENDFOLD (GRIPPERTECH EXT)
;FOLD SPOTTECH EXT
EXT  USERSPOT (S_COMMAND  :IN,SPOT_TYPE  :IN )
;ENDFOLD (SPOTTECH EXT)
;FOLD BASISTECH EXT;%{PE}%MKUKATPBASIS,%CEXT,%VEXT,%P
EXT  BAS (BAS_COMMAND  :IN,REAL  :IN )
DECL INT SUCCESS
;ENDFOLD (BASISTECH EXT)
;FOLD USER EXT;%{E}%MKUKATPUSER,%CEXT,%VEXT,%P
;Make your modifications here

;ENDFOLD (USER EXT)
;ENDFOLD (EXTERNAL DECLARATIONS)

;# ============ START PATH : swp_p13050r4_com_geo_c1 =============
DECL FDAT Fs_lx488={TOOL_NO 1,BASE_NO 1,IPO_FRAME #BASE,POINT2[] " "}
DECL PDAT PP_OLP5={VEL 100.0,ACC 100.0,APO_DIST 100.0,APO_MODE #CDIS}
DECL E6POS Xs_lx488={X -360.817993,Y 965.559021,Z 683.950989,A 93.2594986,B 64.8991013,C -75.3226013,S 2,T 10,E1 4060.29907,E2 0.0,E3 0.0,E4 0.0,E5 0.0,E6 0.0}
DECL FDAT Fswp_60_5140={TOOL_NO 1,BASE_NO 1,IPO_FRAME #BASE,POINT2[] " "}
DECL PDAT PP_OLP7={VEL 100.0,ACC 100.0,APO_DIST 0.0}
DECL SPOT_TYPE SS_OLP1={GUN 1,PAIR #FIRST,RETR #CLO,CLO_TM 0,PGNO1 1,PRESS1 1.0,PGNO2 0,PRESS2 0.0}
DECL E6POS Xswp_60_5140={X 136.687195,Y 902.795288,Z 579.572021,A 83.2147293,B 65.6525803,C -84.4438324,S 2,T 10,E1 4060.30103,E2 0.0,E3 0.0,E4 0.0,E5 0.0,E6 0.0}
DECL FDAT Fs_lx486={TOOL_NO 1,BASE_NO 1,IPO_FRAME #BASE,POINT2[] " "}
DECL PDAT PP_OLP9={VEL 100.0,ACC 100.0,APO_DIST 100.0,APO_MODE #CDIS}
DECL E6POS Xs_lx486={X -360.820007,Y 965.559998,Z 683.950989,A 93.2594986,B 64.8992004,C -75.3226013,S 2,T 10,E1 4060.29907,E2 0.0,E3 0.0,E4 0.0,E5 0.0,E6 0.0}
DECL PDAT PP_OLP10={VEL 100.0,ACC 100.0,APO_DIST 50.0,APO_MODE #CDIS}
DECL FDAT Fswp_60_5118={TOOL_NO 1,BASE_NO 1,IPO_FRAME #BASE,POINT2[] " "}
DECL PDAT PP_OLP12={VEL 100.0,ACC 100.0,APO_DIST 0.0}
DECL SPOT_TYPE SS_OLP2={GUN 1,PAIR #FIRST,RETR #CLO,CLO_TM 0,PGNO1 1,PRESS1 1.0,PGNO2 0,PRESS2 0.0}
DECL E6POS Xswp_60_5118={X 94.381012,Y 322.608704,Z 577.968018,A 0.639736116,B 88.9835663,C -175.218796,S 2,T 10,E1 4060.29199,E2 0.0,E3 0.0,E4 0.0,E5 0.0,E6 0.0}
DECL PDAT PP_OLP14={VEL 100.0,ACC 100.0,APO_DIST 100.0,APO_MODE #CDIS}
DECL PDAT PP_OLP16={VEL 100.0,ACC 100.0,APO_DIST 100.0,APO_MODE #CDIS}
DECL FDAT Fswp_60_5026={TOOL_NO 1,BASE_NO 1,IPO_FRAME #BASE,POINT2[] " "}
DECL PDAT PP_OLP18={VEL 100.0,ACC 100.0,APO_DIST 0.0}
DECL SPOT_TYPE SS_OLP3={GUN 1,PAIR #FIRST,RETR #CLO,CLO_TM 0,PGNO1 1,PRESS1 1.0,PGNO2 0,PRESS2 0.0}
DECL E6POS Xswp_60_5026={X 159.332901,Y 427.524109,Z 4.32035685,A 90.0029831,B -50.8949509,C -90.0011292,S 2,T 42,E1 4060.2771,E2 0.0,E3 0.0,E4 0.0,E5 0.0,E6 0.0}
DECL FDAT Fswp_60_5020={TOOL_NO 1,BASE_NO 1,IPO_FRAME #BASE,POINT2[] " "}
DECL PDAT PP_OLP19={VEL 100.0,ACC 100.0,APO_DIST 0.0}
DECL SPOT_TYPE SS_OLP4={GUN 1,PAIR #FIRST,RETR #CLO,CLO_TM 0,PGNO1 1,PRESS1 1.0,PGNO2 0,PRESS2 0.0}
DECL E6POS Xswp_60_5020={X 158.871796,Y 329.765594,Z 2.61356592,A 90.0077286,B -48.4540215,C -90.0015869,S 2,T 42,E1 4060.2981,E2 0.0,E3 0.0,E4 0.0,E5 0.0,E6 0.0}
DECL FDAT Fswp_60_5016={TOOL_NO 1,BASE_NO 1,IPO_FRAME #BASE,POINT2[] " "}
DECL PDAT PP_OLP20={VEL 100.0,ACC 100.0,APO_DIST 0.0}
DECL SPOT_TYPE SS_OLP5={GUN 1,PAIR #FIRST,RETR #CLO,CLO_TM 0,PGNO1 1,PRESS1 1.0,PGNO2 0,PRESS2 0.0}
DECL E6POS Xswp_60_5016={X 159.657196,Y 262.3927,Z 3.53638506,A 90.0078125,B -48.4543304,C -90.0026169,S 2,T 42,E1 4060.2959,E2 0.0,E3 0.0,E4 0.0,E5 0.0,E6 0.0}
DECL FDAT Fswp_60_5014={TOOL_NO 1,BASE_NO 1,IPO_FRAME #BASE,POINT2[] " "}
DECL PDAT PP_OLP21={VEL 100.0,ACC 100.0,APO_DIST 0.0}
DECL SPOT_TYPE SS_OLP6={GUN 1,PAIR #FIRST,RETR #CLO,CLO_TM 0,PGNO1 1,PRESS1 1.0,PGNO2 0,PRESS2 0.0}
DECL E6POS Xswp_60_5014={X 159.661102,Y 231.6185,Z 3.63049507,A 90.0080414,B -48.4544716,C -90.0028687,S 2,T 42,E1 4060.29712,E2 0.0,E3 0.0,E4 0.0,E5 0.0,E6 0.0}
DECL PDAT PP_OLP22={VEL 100.0,ACC 100.0,APO_DIST 100.0,APO_MODE #CDIS}
DECL FDAT Fs_lx470={TOOL_NO 1,BASE_NO 1,IPO_FRAME #BASE,POINT2[] " "}
DECL PDAT PP_OLP23={VEL 100.0,ACC 100.0,APO_DIST 100.0,APO_MODE #CDIS}
DECL E6POS Xs_lx470={X -243.503998,Y 293.677002,Z -34.257,A 90.0,B -44.5937996,C -90.0,S 2,T 10,E1 4060.29907,E2 0.0,E3 0.0,E4 0.0,E5 0.0,E6 0.0}
DECL PDAT PP_OLP24={VEL 100.0,ACC 100.0,APO_DIST 100.0,APO_MODE #CDIS}
DECL FDAT Flx507={TOOL_NO 1,BASE_NO 1,IPO_FRAME #BASE,POINT2[] " "}
DECL PDAT PP_OLP25={VEL 100.0,ACC 100.0,APO_DIST 100.0,APO_MODE #CDIS}
DECL E6POS Xlx507={X -11.6990004,Y 1057.32996,Z -233.384003,A 68.1399002,B -45.7775993,C -90.0,S 2,T 10,E1 4060.29907,E2 0.0,E3 0.0,E4 0.0,E5 0.0,E6 0.0}
DECL PDAT PP_OLP26={VEL 100.0,ACC 100.0,APO_DIST 100.0,APO_MODE #CDIS}
DECL FDAT Fswp_60_5042={TOOL_NO 1,BASE_NO 1,IPO_FRAME #BASE,POINT2[] " "}
DECL PDAT PP_OLP27={VEL 100.0,ACC 100.0,APO_DIST 0.0}
DECL SPOT_TYPE SS_OLP7={GUN 1,PAIR #FIRST,RETR #CLO,CLO_TM 0,PGNO1 1,PRESS1 1.0,PGNO2 0,PRESS2 0.0}
DECL E6POS Xswp_60_5042={X 176.981293,Y 1036.93799,Z -181.563095,A 68.1404114,B -45.7783699,C -90.0011597,S 2,T 10,E1 4060.30005,E2 0.0,E3 0.0,E4 0.0,E5 0.0,E6 0.0}
DECL FDAT Fswp_60_5040={TOOL_NO 1,BASE_NO 1,IPO_FRAME #BASE,POINT2[] " "}
DECL PDAT PP_OLP28={VEL 100.0,ACC 100.0,APO_DIST 0.0}
DECL SPOT_TYPE SS_OLP8={GUN 1,PAIR #FIRST,RETR #CLO,CLO_TM 0,PGNO1 1,PRESS1 1.0,PGNO2 0,PRESS2 0.0}
DECL E6POS Xswp_60_5040={X 172.178604,Y 1008.79102,Z -183.401794,A 176.628098,B -88.2014084,C 167.694305,S 2,T 10,E1 4060.30103,E2 0.0,E3 0.0,E4 0.0,E5 0.0,E6 0.0}
DECL FDAT Fswp_60_5038={TOOL_NO 1,BASE_NO 1,IPO_FRAME #BASE,POINT2[] " "}
DECL PDAT PP_OLP29={VEL 100.0,ACC 100.0,APO_DIST 0.0}
DECL SPOT_TYPE SS_OLP9={GUN 1,PAIR #FIRST,RETR #CLO,CLO_TM 0,PGNO1 1,PRESS1 1.0,PGNO2 0,PRESS2 0.0}
DECL E6POS Xswp_60_5038={X 164.622696,Y 982.143127,Z -183.500595,A -120.116699,B -89.1609726,C 109.444,S 2,T 10,E1 4060.29907,E2 0.0,E3 0.0,E4 0.0,E5 0.0,E6 0.0}
DECL FDAT Fswp_60_5036={TOOL_NO 1,BASE_NO 1,IPO_FRAME #BASE,POINT2[] " "}
DECL SPOT_TYPE SS_OLP10={GUN 1,PAIR #FIRST,RETR #CLO,CLO_TM 0,PGNO1 1,PRESS1 1.0,PGNO2 0,PRESS2 0.0}
DECL E6POS Xswp_60_5036={X 179.731094,Y 901.85553,Z -137.682495,A -105.0299,B -89.9987488,C 105.028702,S 2,T 42,E1 4060.29907,E2 0.0,E3 0.0,E4 0.0,E5 0.0,E6 0.0}
DECL FDAT Fswp_60_5028={TOOL_NO 1,BASE_NO 1,IPO_FRAME #BASE,POINT2[] " "}
DECL PDAT PP_OLP32={VEL 100.0,ACC 100.0,APO_DIST 0.0}
DECL SPOT_TYPE SS_OLP11={GUN 1,PAIR #FIRST,RETR #CLO,CLO_TM 0,PGNO1 1,PRESS1 1.0,PGNO2 0,PRESS2 0.0}
DECL E6POS Xswp_60_5028={X 182.583893,Y 794.820129,Z -47.8096008,A -163.747406,B -89.5717773,C 163.750702,S 2,T 42,E1 4060.29395,E2 0.0,E3 0.0,E4 0.0,E5 0.0,E6 0.0}
DECL FDAT Fs_lx464={TOOL_NO 1,BASE_NO 1,IPO_FRAME #BASE,POINT2[] " "}
DECL PDAT PP_OLP33={VEL 100.0,ACC 100.0,APO_DIST 100.0,APO_MODE #CDIS}
DECL E6POS Xs_lx464={X 178.498993,Y 805.025024,Z -118.82,A 0.0,B -90.0,C 0.0,S 2,T 42,E1 4060.29907,E2 0.0,E3 0.0,E4 0.0,E5 0.0,E6 0.0}
DECL PDAT PP_OLP34={VEL 100.0,ACC 100.0,APO_DIST 100.0,APO_MODE #CDIS}
DECL SPOT_TYPE SS_OLP12={GUN 1,PAIR #FIRST,RETR #CLO,CLO_TM 0,PGNO1 1,PRESS1 1.0,PGNO2 0,PRESS2 0.0}
DECL FDAT Fswp_60_5203={TOOL_NO 1,BASE_NO 1,IPO_FRAME #BASE,POINT2[] " "}
DECL SPOT_TYPE SS_OLP13={GUN 1,PAIR #FIRST,RETR #CLO,CLO_TM 0,PGNO1 1,PRESS1 1.0,PGNO2 0,PRESS2 0.0}
DECL E6POS Xswp_60_5203={X 156.1819,Y 485.568604,Z 388.023712,A 90.0274734,B -54.6427803,C -86.9009323,S 2,T 10,E1 4060.31592,E2 0.0,E3 0.0,E4 0.0,E5 0.0,E6 0.0}
DECL FDAT Fswp_60_5195={TOOL_NO 1,BASE_NO 1,IPO_FRAME #BASE,POINT2[] " "}
DECL SPOT_TYPE SS_OLP14={GUN 1,PAIR #FIRST,RETR #CLO,CLO_TM 0,PGNO1 1,PRESS1 1.0,PGNO2 0,PRESS2 0.0}
DECL E6POS Xswp_60_5195={X 161.142303,Y 202.515198,Z 386.019104,A -88.2071686,B -36.5904808,C 88.8797302,S 2,T 10,E1 4060.31396,E2 0.0,E3 0.0,E4 0.0,E5 0.0,E6 0.0}
DECL FDAT Fswp_60_5190={TOOL_NO 1,BASE_NO 1,IPO_FRAME #BASE,POINT2[] " "}
DECL SPOT_TYPE SS_OLP15={GUN 1,PAIR #FIRST,RETR #CLO,CLO_TM 0,PGNO1 1,PRESS1 1.0,PGNO2 0,PRESS2 0.0}
DECL E6POS Xswp_60_5190={X 161.480301,Y 148.9478,Z 280.717194,A -89.3926468,B -1.94816995,C 88.6738968,S 2,T 10,E1 4060.31494,E2 0.0,E3 0.0,E4 0.0,E5 0.0,E6 0.0}
DECL FDAT Fswp_60_5218={TOOL_NO 1,BASE_NO 1,IPO_FRAME #BASE,POINT2[] " "}
DECL SPOT_TYPE SS_OLP16={GUN 1,PAIR #FIRST,RETR #CLO,CLO_TM 0,PGNO1 1,PRESS1 1.0,PGNO2 0,PRESS2 0.0}
DECL E6POS Xswp_60_5218={X 164.738403,Y 122.212402,Z 106.1138,A -90.9965591,B 31.5576591,C 87.71698,S 2,T 10,E1 4060.31396,E2 0.0,E3 0.0,E4 0.0,E5 0.0,E6 0.0}
DECL PDAT PP_OLP52={VEL 100.0,ACC 100.0,APO_DIST 100.0,APO_MODE #CDIS}
DECL SPOT_TYPE SS_OLP17={GUN 1,PAIR #FIRST,RETR #CLO,CLO_TM 0,PGNO1 1,PRESS1 1.0,PGNO2 0,PRESS2 0.0}
DECL SPOT_TYPE SS_OLP18={GUN 1,PAIR #FIRST,RETR #CLO,CLO_TM 0,PGNO1 1,PRESS1 1.0,PGNO2 0,PRESS2 0.0}
DECL SPOT_TYPE SS_OLP19={GUN 1,PAIR #FIRST,RETR #CLO,CLO_TM 0,PGNO1 1,PRESS1 1.0,PGNO2 0,PRESS2 0.0}
DECL FDAT Fswp_60_5066={TOOL_NO 1,BASE_NO 1,IPO_FRAME #BASE,POINT2[] " "}
DECL SPOT_TYPE SS_OLP20={GUN 1,PAIR #FIRST,RETR #CLO,CLO_TM 0,PGNO1 1,PRESS1 1.0,PGNO2 0,PRESS2 0.0}
DECL E6POS Xswp_60_5066={X 151.353302,Y 626.425415,Z 250.5159,A -92.1195831,B 18.5633907,C 91.8053436,S 2,T 10,E1 4060.30591,E2 0.0,E3 0.0,E4 0.0,E5 0.0,E6 0.0}
DECL PDAT PP_OLP59={VEL 100.0,ACC 100.0,APO_DIST 20.0,APO_MODE #CDIS}
DECL PDAT PP_OLP60={VEL 100.0,ACC 100.0,APO_DIST 20.0,APO_MODE #CDIS}
DECL PDAT PP_OLP61={VEL 100.0,ACC 100.0,APO_DIST 20.0,APO_MODE #CDIS}
DECL FDAT Fswp_60_5076={TOOL_NO 1,BASE_NO 1,IPO_FRAME #BASE,POINT2[] " "}
DECL PDAT PP_OLP63={VEL 100.0,ACC 100.0,APO_DIST 0.0}
DECL SPOT_TYPE SS_OLP21={GUN 1,PAIR #FIRST,RETR #CLO,CLO_TM 0,PGNO1 1,PRESS1 1.0,PGNO2 0,PRESS2 0.0}
DECL E6POS Xswp_60_5076={X 154.796707,Y 782.258972,Z 101.740097,A 87.1909637,B 70.1359329,C -93.0589066,S 2,T 10,E1 4060.29199,E2 0.0,E3 0.0,E4 0.0,E5 0.0,E6 0.0}
DECL PDAT PP_OLP64={VEL 100.0,ACC 100.0,APO_DIST 100.0,APO_MODE #CDIS}
DECL SPOT_TYPE SS_OLP22={GUN 1,PAIR #FIRST,RETR #CLO,CLO_TM 0,PGNO1 1,PRESS1 1.0,PGNO2 0,PRESS2 0.0}
DECL PDAT PP_OLP69={VEL 100.0,ACC 100.0,APO_DIST 100.0,APO_MODE #CDIS}
DECL PDAT PP_OLP72={VEL 100.0,ACC 100.0,APO_DIST 100.0,APO_MODE #CDIS}
DECL FDAT Fswp_60_5626={TOOL_NO 1,BASE_NO 1,IPO_FRAME #BASE,POINT2[] " "}
DECL PDAT PP_OLP73={VEL 100.0,ACC 100.0,APO_DIST 0.0}
DECL SPOT_TYPE SS_OLP23={GUN 1,PAIR #FIRST,RETR #CLO,CLO_TM 0,PGNO1 1,PRESS1 1.0,PGNO2 0,PRESS2 0.0}
DECL E6POS Xswp_60_5626={X 634.33252,Y 1098.11096,Z 1372.00806,A -179.633102,B -69.9991837,C 90.5753021,S 2,T 2,E1 5254.49902,E2 0.0,E3 0.0,E4 0.0,E5 0.0,E6 0.0}
DECL FDAT Fswp_60_5640={TOOL_NO 1,BASE_NO 1,IPO_FRAME #BASE,POINT2[] " "}
DECL PDAT PP_OLP74={VEL 100.0,ACC 100.0,APO_DIST 0.0}
DECL SPOT_TYPE SS_OLP24={GUN 1,PAIR #FIRST,RETR #CLO,CLO_TM 0,PGNO1 1,PRESS1 1.0,PGNO2 0,PRESS2 0.0}
DECL E6POS Xswp_60_5640={X 731.3703,Y 1097.53699,Z 1377.57104,A 0.929155171,B -80.0200806,C -89.9900208,S 2,T 2,E1 5254.5,E2 0.0,E3 0.0,E4 0.0,E5 0.0,E6 0.0}
DECL PDAT PP_OLP75={VEL 100.0,ACC 100.0,APO_DIST 100.0,APO_MODE #CDIS}
DECL PDAT PP_OLP76={VEL 100.0,ACC 100.0,APO_DIST 100.0,APO_MODE #CDIS}
DECL PDAT PP_OLP77={VEL 100.0,ACC 100.0,APO_DIST 50.0,APO_MODE #CDIS}
DECL PDAT PP_OLP78={VEL 100.0,ACC 100.0,APO_DIST 50.0,APO_MODE #CDIS}
DECL FDAT Fswp_60_5060={TOOL_NO 1,BASE_NO 1,IPO_FRAME #BASE,POINT2[] " "}
DECL PDAT PP_OLP79={VEL 100.0,ACC 100.0,APO_DIST 0.0}
DECL SPOT_TYPE SS_OLP25={GUN 1,PAIR #FIRST,RETR #CLO,CLO_TM 0,PGNO1 1,PRESS1 1.0,PGNO2 0,PRESS2 0.0}
DECL E6POS Xswp_60_5060={X 440.014313,Y 1093.56006,Z -44.92976,A -177.803696,B 33.6436501,C 90.0005798,S 2,T 34,E1 5251.46289,E2 0.0,E3 0.0,E4 0.0,E5 0.0,E6 0.0}
DECL PDAT PP_OLP80={VEL 100.0,ACC 100.0,APO_DIST 50.0,APO_MODE #CDIS}
DECL PDAT PP_OLP81={VEL 100.0,ACC 100.0,APO_DIST 50.0,APO_MODE #CDIS}
DECL PDAT PP_OLP82={VEL 100.0,ACC 100.0,APO_DIST 100.0,APO_MODE #CDIS}
DECL FDAT Fswp_60_5056={TOOL_NO 1,BASE_NO 1,IPO_FRAME #BASE,POINT2[] " "}
DECL PDAT PP_OLP85={VEL 100.0,ACC 100.0,APO_DIST 0.0}
DECL SPOT_TYPE SS_OLP26={GUN 1,PAIR #FIRST,RETR #CLO,CLO_TM 0,PGNO1 1,PRESS1 1.0,PGNO2 0,PRESS2 0.0}
DECL E6POS Xswp_60_5056={X 372.068909,Y 1092.44397,Z -181.150497,A 178.998093,B -2.52557802,C 89.9496765,S 2,T 34,E1 5252.67188,E2 0.0,E3 0.0,E4 0.0,E5 0.0,E6 0.0}
DECL FDAT Fswp_60_5058={TOOL_NO 1,BASE_NO 1,IPO_FRAME #BASE,POINT2[] " "}
DECL PDAT PP_OLP86={VEL 100.0,ACC 100.0,APO_DIST 0.0}
DECL SPOT_TYPE SS_OLP27={GUN 1,PAIR #FIRST,RETR #CLO,CLO_TM 0,PGNO1 1,PRESS1 1.0,PGNO2 0,PRESS2 0.0}
DECL E6POS Xswp_60_5058={X 404.384796,Y 1091.41699,Z -160.593002,A 178.922501,B -10.25455,C 90.7412491,S 2,T 34,E1 5253.80078,E2 0.0,E3 0.0,E4 0.0,E5 0.0,E6 0.0}
DECL PDAT PP_OLP88={VEL 100.0,ACC 100.0,APO_DIST 100.0,APO_MODE #CDIS}
DECL PDAT PP_OLP89={VEL 100.0,ACC 100.0,APO_DIST 100.0,APO_MODE #CDIS}
DECL FDAT Fswp_60_5424={TOOL_NO 1,BASE_NO 1,IPO_FRAME #BASE,POINT2[] " "}
DECL PDAT PP_OLP91={VEL 100.0,ACC 100.0,APO_DIST 0.0}
DECL SPOT_TYPE SS_OLP28={GUN 1,PAIR #FIRST,RETR #CLO,CLO_TM 0,PGNO1 1,PRESS1 1.0,PGNO2 0,PRESS2 0.0}
DECL E6POS Xswp_60_5424={X 1302.37805,Y 1186.15405,Z -56.5237999,A -0.546349108,B -50.1205597,C -90.0004196,S 2,T 2,E1 5251.78613,E2 0.0,E3 0.0,E4 0.0,E5 0.0,E6 0.0}
DECL PDAT PP_OLP92={VEL 100.0,ACC 100.0,APO_DIST 100.0,APO_MODE #CDIS}
DECL PDAT PP_OLP93={VEL 100.0,ACC 100.0,APO_DIST 100.0,APO_MODE #CDIS}
DECL PDAT PP_OLP96={VEL 100.0,ACC 100.0,APO_DIST 100.0,APO_MODE #CDIS}
DECL PDAT PP_OLP97={VEL 100.0,ACC 100.0,APO_DIST 20.0,APO_MODE #CDIS}
DECL FDAT Fswp_60_5430={TOOL_NO 1,BASE_NO 1,IPO_FRAME #BASE,POINT2[] " "}
DECL PDAT PP_OLP100={VEL 100.0,ACC 100.0,APO_DIST 0.0}
DECL SPOT_TYPE SS_OLP29={GUN 1,PAIR #FIRST,RETR #CLO,CLO_TM 0,PGNO1 1,PRESS1 1.0,PGNO2 0,PRESS2 0.0}
DECL E6POS Xswp_60_5430={X 1286.38098,Y 1123.69702,Z 5.72508383,A -0.644820571,B 48.2571411,C -90.0793915,S 2,T 2,E1 6178.22119,E2 0.0,E3 0.0,E4 0.0,E5 0.0,E6 0.0}
DECL FDAT Fswp_60_5432={TOOL_NO 1,BASE_NO 1,IPO_FRAME #BASE,POINT2[] " "}
DECL PDAT PP_OLP101={VEL 100.0,ACC 100.0,APO_DIST 0.0}
DECL SPOT_TYPE SS_OLP30={GUN 1,PAIR #FIRST,RETR #CLO,CLO_TM 0,PGNO1 1,PRESS1 1.0,PGNO2 0,PRESS2 0.0}
DECL E6POS Xswp_60_5432={X 1304.38,Y 1123.71106,Z 21.1026192,A -0.644798875,B 48.25737,C -90.0797424,S 2,T 2,E1 6217.10498,E2 0.0,E3 0.0,E4 0.0,E5 0.0,E6 0.0}
DECL FDAT Fswp_60_5434={TOOL_NO 1,BASE_NO 1,IPO_FRAME #BASE,POINT2[] " "}
DECL PDAT PP_OLP102={VEL 100.0,ACC 100.0,APO_DIST 0.0}
DECL SPOT_TYPE SS_OLP31={GUN 1,PAIR #FIRST,RETR #CLO,CLO_TM 0,PGNO1 1,PRESS1 1.0,PGNO2 0,PRESS2 0.0}
DECL E6POS Xswp_60_5434={X 1288.31995,Y 1122.44202,Z 30.7160091,A -0.641988695,B 48.2577095,C -90.0761871,S 2,T 2,E1 6172.71387,E2 0.0,E3 0.0,E4 0.0,E5 0.0,E6 0.0}
DECL FDAT Fswp_60_5436={TOOL_NO 1,BASE_NO 1,IPO_FRAME #BASE,POINT2[] " "}
DECL PDAT PP_OLP105={VEL 100.0,ACC 100.0,APO_DIST 0.0}
DECL SPOT_TYPE SS_OLP32={GUN 1,PAIR #FIRST,RETR #CLO,CLO_TM 0,PGNO1 1,PRESS1 1.0,PGNO2 0,PRESS2 0.0}
DECL E6POS Xswp_60_5436={X 1304.93005,Y 1120.12903,Z 80.8903885,A -0.630691886,B 29.8777504,C -90.0939484,S 2,T 2,E1 6169.68115,E2 0.0,E3 0.0,E4 0.0,E5 0.0,E6 0.0}
DECL FDAT Fswp_60_5438={TOOL_NO 1,BASE_NO 1,IPO_FRAME #BASE,POINT2[] " "}
DECL PDAT PP_OLP107={VEL 100.0,ACC 100.0,APO_DIST 0.0}
DECL SPOT_TYPE SS_OLP33={GUN 1,PAIR #FIRST,RETR #CLO,CLO_TM 0,PGNO1 1,PRESS1 1.0,PGNO2 0,PRESS2 0.0}
DECL E6POS Xswp_60_5438={X 1335.14502,Y 1125.09802,Z 99.5109024,A -0.583152175,B 19.4271107,C -90.0527191,S 2,T 2,E1 5977.15283,E2 0.0,E3 0.0,E4 0.0,E5 0.0,E6 0.0}
DECL FDAT Fswp_60_5440={TOOL_NO 1,BASE_NO 1,IPO_FRAME #BASE,POINT2[] " "}
DECL PDAT PP_OLP108={VEL 100.0,ACC 100.0,APO_DIST 0.0}
DECL SPOT_TYPE SS_OLP34={GUN 1,PAIR #FIRST,RETR #CLO,CLO_TM 0,PGNO1 1,PRESS1 1.0,PGNO2 0,PRESS2 0.0}
DECL E6POS Xswp_60_5440={X 1334.10596,Y 1122.04004,Z 140.932205,A -0.565891325,B -2.25514102,C -90.0501328,S 2,T 2,E1 5826.48584,E2 0.0,E3 0.0,E4 0.0,E5 0.0,E6 0.0}
DECL PDAT PP_OLP109={VEL 100.0,ACC 100.0,APO_DIST 100.0,APO_MODE #CDIS}
DECL PDAT PP_OLP110={VEL 100.0,ACC 100.0,APO_DIST 100.0,APO_MODE #CDIS}
DECL PDAT PP_OLP111={VEL 100.0,ACC 100.0,APO_DIST 100.0,APO_MODE #CDIS}
DECL PDAT PP_OLP112={VEL 100.0,ACC 100.0,APO_DIST 100.0,APO_MODE #CDIS}
DECL PDAT PP_OLP113={VEL 100.0,ACC 100.0,APO_DIST 0.0,APO_MODE #CDIS}
DECL BASIS_SUGG_T LAST_BASIS={POINT1[] "P0                      ",POINT2[] "P0                      ",CP_PARAMS[] "CPDAT0                  ",PTP_PARAMS[] "PDAT0                   ",CONT[] "                        ",CP_VEL[] "2.0                     ",PTP_VEL[] " 100                    ",SYNC_PARAMS[] "SYNCDAT                 ",SPL_NAME[] "S0                      "}
DECL FDAT FXs_lx487={TOOL_NO 1,BASE_NO 1,IPO_FRAME #BASE,POINT2[] " ",TQ_STATE FALSE}
DECL E6POS XXS_LX487={X 142.0215,Y 865.563782,Z 629.299988,A 92.7790527,B 65.0505371,C -75.8403931,S 2,T 10,E1 4060.29395,E2 0.0,E3 0.0,E4 0.0,E5 0.0,E6 0.0}
DECL PDAT PPDAT2={VEL 100.0,ACC 100.0,APO_DIST 100.0,APO_MODE #CDIS}
DECL E6POS XXS_LX502={X 142.021301,Y 865.560791,Z 629.294983,A 92.7791138,B 65.0502167,C -75.8401871,S 2,T 10,E1 4060.29395,E2 0.0,E3 0.0,E4 0.0,E5 0.0,E6 0.0}
DECL FDAT FXs_lx502={TOOL_NO 1,BASE_NO 1,IPO_FRAME #BASE,POINT2[] " ",TQ_STATE FALSE}
DECL PDAT PPDAT6={VEL 100.0,ACC 100.0,APO_DIST 100.0,APO_MODE #CDIS}
DECL E6POS XXS_LX484={X -406.284088,Y 364.974487,Z 582.284119,A -59.6039505,B 89.6699677,C 128.917496,S 2,T 10,E1 4060.2981,E2 0.0,E3 0.0,E4 0.0,E5 0.0,E6 0.0}
DECL FDAT FXs_lx484={TOOL_NO 1,BASE_NO 1,IPO_FRAME #BASE,POINT2[] " ",TQ_STATE FALSE}
DECL E6POS XXS_LX504={X 102.534103,Y 321.186096,Z 604.033508,A 152.166595,B 89.932457,C -19.8392105,S 2,T 10,E1 4060.30005,E2 0.0,E3 0.0,E4 0.0,E5 0.0,E6 0.0}
DECL FDAT FXs_lx504={TOOL_NO 1,BASE_NO 1,IPO_FRAME #BASE,POINT2[] " ",TQ_STATE FALSE}
DECL PDAT PPDAT8={VEL 100.0,ACC 100.0,APO_DIST 50.0,APO_MODE #CDIS}
DECL E6POS XXS_LX506={X 101.603203,Y 324.702209,Z 606.954773,A -105.589798,B 89.533989,C 82.46315,S 2,T 10,E1 4060.29907,E2 0.0,E3 0.0,E4 0.0,E5 0.0,E6 0.0}
DECL FDAT FXs_lx506={TOOL_NO 1,BASE_NO 1,IPO_FRAME #BASE,POINT2[] " ",TQ_STATE FALSE}
DECL PDAT PPDAT10={VEL 100.0,ACC 100.0,APO_DIST 100.0,APO_MODE #CDIS}
DECL E6POS XXS_LX482={X -401.920288,Y 344.626587,Z 598.098022,A -123.613403,B 89.7013168,C 73.3319473,S 2,T 10,E1 4060.2981,E2 0.0,E3 0.0,E4 0.0,E5 0.0,E6 0.0}
DECL FDAT FXs_lx482={TOOL_NO 1,BASE_NO 1,IPO_FRAME #BASE,POINT2[] " ",TQ_STATE FALSE}
DECL E6POS XXS_LX510={X 164.903503,Y 407.34549,Z -24.669241,A 90.0030136,B -50.8949699,C -90.0012512,S 2,T 42,E1 4060.2771,E2 0.0,E3 0.0,E4 0.0,E5 0.0,E6 0.0}
DECL FDAT FXs_lx510={TOOL_NO 1,BASE_NO 1,IPO_FRAME #BASE,POINT2[] " ",TQ_STATE FALSE}
DECL PDAT PPDAT14={VEL 100.0,ACC 100.0,APO_DIST 100.0,APO_MODE #CDIS}
DECL E6POS XXS_LX469={X 176.571396,Y 282.161896,Z -22.7473507,A 89.9942474,B -44.593441,C -89.9960175,S 2,T 42,E1 4060.30103,E2 0.0,E3 0.0,E4 0.0,E5 0.0,E6 0.0}
DECL FDAT FXs_lx469={TOOL_NO 1,BASE_NO 1,IPO_FRAME #BASE,POINT2[] " ",TQ_STATE FALSE}
DECL E6POS XXS_LX468={X -247.606094,Y 804.985718,Z -118.853699,A 19.7734299,B -89.9986496,C -19.7741909,S 2,T 42,E1 4060.29907,E2 0.0,E3 0.0,E4 0.0,E5 0.0,E6 0.0}
DECL FDAT FXs_lx468={TOOL_NO 1,BASE_NO 1,IPO_FRAME #BASE,POINT2[] " ",TQ_STATE FALSE}
DECL E6POS XXS_LX512={X 180.2099,Y 1013.57098,Z -191.423492,A -25.3134308,B -87.7871933,C 9.87290573,S 2,T 10,E1 4060.29907,E2 0.0,E3 0.0,E4 0.0,E5 0.0,E6 0.0}
DECL FDAT FXs_lx512={TOOL_NO 1,BASE_NO 1,IPO_FRAME #BASE,POINT2[] " ",TQ_STATE FALSE}
DECL PDAT PPDAT16={VEL 100.0,ACC 100.0,APO_DIST 100.0,APO_MODE #CDIS}
DECL E6POS XXS_LX514={X 200.297501,Y 951.728088,Z -170.494797,A -120.180603,B -89.1640396,C 109.508102,S 2,T 10,E1 4060.2981,E2 0.0,E3 0.0,E4 0.0,E5 0.0,E6 0.0}
DECL FDAT FXs_lx514={TOOL_NO 1,BASE_NO 1,IPO_FRAME #BASE,POINT2[] " ",TQ_STATE FALSE}
DECL PDAT PPDAT18={VEL 100.0,ACC 100.0,APO_DIST 100.0,APO_MODE #CDIS}
DECL E6POS XXS_LX465={X -260.471985,Y 805.001709,Z -118.772697,A 138.775497,B -89.9979477,C -138.775497,S 2,T 42,E1 4060.31104,E2 0.0,E3 0.0,E4 0.0,E5 0.0,E6 0.0}
DECL FDAT FXs_lx465={TOOL_NO 1,BASE_NO 1,IPO_FRAME #BASE,POINT2[] " ",TQ_STATE FALSE}
DECL E6POS XXLX510={X 198.537292,Y 907.492188,Z 358.6026,A 89.3582687,B -28.1856194,C -88.5561295,S 2,T 10,E1 4060.30005,E2 0.0,E3 0.0,E4 0.0,E5 0.0,E6 0.0}
DECL FDAT FXlx510={TOOL_NO 1,BASE_NO 1,IPO_FRAME #BASE,POINT2[] " ",TQ_STATE FALSE}
DECL E6POS XXS_LX456={X -359.326691,Y 798.908997,Z 114.357002,A 87.1922531,B 70.1376114,C -93.0576477,S 2,T 10,E1 4060.30396,E2 0.0,E3 0.0,E4 0.0,E5 0.0,E6 0.0}
DECL FDAT FXs_lx456={TOOL_NO 1,BASE_NO 1,IPO_FRAME #BASE,POINT2[] " ",TQ_STATE FALSE}
DECL E6POS XXS_LX455={X -1161.73706,Y 2536.57007,Z -258.942688,A -75.5931015,B -3.65610003,C -1.19887197,S 2,T 2,E1 4060.30005,E2 0.0,E3 0.0,E4 0.0,E5 0.0,E6 0.0}
DECL FDAT FXs_lx455={TOOL_NO 1,BASE_NO 1,IPO_FRAME #BASE,POINT2[] " ",TQ_STATE FALSE}
DECL E6POS XXS_LX449={X 694.406311,Y 1082.60999,Z 1348.03699,A 1.31180894,B -80.1795273,C -90.3731537,S 2,T 2,E1 5254.49707,E2 0.0,E3 0.0,E4 0.0,E5 0.0,E6 0.0}
DECL FDAT FXs_lx449={TOOL_NO 1,BASE_NO 1,IPO_FRAME #BASE,POINT2[] " ",TQ_STATE FALSE}
DECL E6POS XXS_LX447={X 711.179504,Y 1091.54102,Z 1352.49304,A 0.941952884,B -85.4546738,C -90.002861,S 2,T 2,E1 5254.49902,E2 0.0,E3 0.0,E4 0.0,E5 0.0,E6 0.0}
DECL FDAT FXs_lx447={TOOL_NO 1,BASE_NO 1,IPO_FRAME #BASE,POINT2[] " ",TQ_STATE FALSE}
DECL E6POS XXS_LX448={X 697.610718,Y 1743.328,Z 1372.71704,A 0.930606484,B -81.3462601,C -89.9841232,S 2,T 2,E1 5254.5,E2 0.0,E3 0.0,E4 0.0,E5 0.0,E6 0.0}
DECL FDAT FXs_lx448={TOOL_NO 1,BASE_NO 1,IPO_FRAME #BASE,POINT2[] " ",TQ_STATE FALSE}
DECL E6POS XXS_LX446={X 371.822113,Y 1600.547,Z 7.65825987,A -177.905502,B 2.046278,C 91.1621094,S 2,T 34,E1 5251.48584,E2 0.0,E3 0.0,E4 0.0,E5 0.0,E6 0.0}
DECL FDAT FXs_lx446={TOOL_NO 1,BASE_NO 1,IPO_FRAME #BASE,POINT2[] " ",TQ_STATE FALSE}
DECL E6POS XXS_LX445={X 424.494812,Y 1084.04297,Z 14.3757401,A -177.9991,B 7.22483206,C 89.9997635,S 2,T 34,E1 5251.43408,E2 0.0,E3 0.0,E4 0.0,E5 0.0,E6 0.0}
DECL FDAT FXs_lx445={TOOL_NO 1,BASE_NO 1,IPO_FRAME #BASE,POINT2[] " ",TQ_STATE FALSE}
DECL E6POS XXS_LX442={X 424.496094,Y 1084.04297,Z 14.3774099,A -177.998993,B 7.22493505,C 89.9998398,S 2,T 34,E1 5251.43408,E2 0.0,E3 0.0,E4 0.0,E5 0.0,E6 0.0}
DECL FDAT FXs_lx442={TOOL_NO 1,BASE_NO 1,IPO_FRAME #BASE,POINT2[] " ",TQ_STATE FALSE}
DECL E6POS XXS_LX444={X 371.822113,Y 1600.547,Z 7.65825987,A -177.905502,B 2.046278,C 91.1621094,S 2,T 34,E1 5251.48584,E2 0.0,E3 0.0,E4 0.0,E5 0.0,E6 0.0}
DECL FDAT FXs_lx444={TOOL_NO 1,BASE_NO 1,IPO_FRAME #BASE,POINT2[] " ",TQ_STATE FALSE}
DECL E6POS XXS_LX520={X 449.010986,Y 1058.51904,Z -203.744797,A -179.592407,B -0.526983023,C 88.4325333,S 2,T 34,E1 5247.50293,E2 0.0,E3 0.0,E4 0.0,E5 0.0,E6 0.0}
DECL FDAT FXs_lx520={TOOL_NO 1,BASE_NO 1,IPO_FRAME #BASE,POINT2[] " ",TQ_STATE FALSE}
DECL PDAT PPDAT24={VEL 100.0,ACC 100.0,APO_DIST 100.0,APO_MODE #CDIS}
DECL E6POS XXS_LX521={X 401.931091,Y 1092.10706,Z -181.568497,A 179.003494,B -2.52484202,C 89.9398193,S 2,T 34,E1 5252.71582,E2 0.0,E3 0.0,E4 0.0,E5 0.0,E6 0.0}
DECL FDAT FXs_lx521={TOOL_NO 1,BASE_NO 1,IPO_FRAME #BASE,POINT2[] " ",TQ_STATE FALSE}
DECL PDAT PPDAT25={VEL 100.0,ACC 100.0,APO_DIST 100.0,APO_MODE #CDIS}
DECL E6POS XXS_LX522={X 448.946808,Y 1058.54504,Z -203.671799,A -179.594101,B -0.524964929,C 88.4331894,S 2,T 34,E1 5254.93994,E2 0.0,E3 0.0,E4 0.0,E5 0.0,E6 0.0}
DECL FDAT FXs_lx522={TOOL_NO 1,BASE_NO 1,IPO_FRAME #BASE,POINT2[] " ",TQ_STATE FALSE}
DECL PDAT PPDAT26={VEL 100.0,ACC 100.0,APO_DIST 100.0,APO_MODE #CDIS}
DECL E6POS XXS_LX439={X 1275.48706,Y 1356.73999,Z -29.0001392,A -10.9303904,B -49.6493797,C -82.047081,S 2,T 2,E1 5253.81494,E2 0.0,E3 0.0,E4 0.0,E5 0.0,E6 0.0}
DECL FDAT FXs_lx439={TOOL_NO 1,BASE_NO 1,IPO_FRAME #BASE,POINT2[] " ",TQ_STATE FALSE}
DECL E6POS XXS_LX524={X 1273.81299,Y 1177.25403,Z -109.4813,A -0.543687284,B -50.1182213,C -90.0044937,S 2,T 2,E1 5254.08496,E2 0.0,E3 0.0,E4 0.0,E5 0.0,E6 0.0}
DECL FDAT FXs_lx524={TOOL_NO 1,BASE_NO 1,IPO_FRAME #BASE,POINT2[] " ",TQ_STATE FALSE}
DECL PDAT PPDAT28={VEL 100.0,ACC 100.0,APO_DIST 20.0,APO_MODE #CDIS}
DECL E6POS XXS_LX434={X 1246.71497,Y 1183.89099,Z -102.509003,A -0.541095018,B -50.1177406,C -89.9982834,S 2,T 2,E1 5254.50391,E2 0.0,E3 0.0,E4 0.0,E5 0.0,E6 0.0}
DECL FDAT FXs_lx434={TOOL_NO 1,BASE_NO 1,IPO_FRAME #BASE,POINT2[] " ",TQ_STATE FALSE}
DECL E6POS XXS_LX525={X 1310.61304,Y 1545.06897,Z 103.151604,A -0.480830699,B -25.6063499,C -90.1753235,S 2,T 2,E1 5255.80176,E2 0.0,E3 0.0,E4 0.0,E5 0.0,E6 0.0}
DECL FDAT FXs_lx525={TOOL_NO 1,BASE_NO 1,IPO_FRAME #BASE,POINT2[] " ",TQ_STATE FALSE}
DECL PDAT PPDAT29={VEL 100.0,ACC 100.0,APO_DIST 100.0,APO_MODE #CDIS}
DECL E6POS XXS_LX526={X 1300.245,Y 1113.05396,Z 132.605804,A -0.57613349,B -13.6800003,C -89.9665985,S 2,T 2,E1 5571.7251,E2 0.0,E3 0.0,E4 0.0,E5 0.0,E6 0.0}
DECL FDAT FXs_lx526={TOOL_NO 1,BASE_NO 1,IPO_FRAME #BASE,POINT2[] " ",TQ_STATE FALSE}
DECL PDAT PPDAT30={VEL 100.0,ACC 100.0,APO_DIST 100.0,APO_MODE #CDIS}
DECL E6POS XXS_LX527={X 1292.80896,Y 1157.88098,Z 128.380295,A -0.5843454,B -17.4577408,C -89.9393997,S 2,T 2,E1 5253.43018,E2 0.0,E3 0.0,E4 0.0,E5 0.0,E6 0.0}
DECL FDAT FXs_lx527={TOOL_NO 1,BASE_NO 1,IPO_FRAME #BASE,POINT2[] " ",TQ_STATE FALSE}
DECL PDAT PPDAT31={VEL 100.0,ACC 100.0,APO_DIST 100.0,APO_MODE #CDIS}
DECL E6POS XXS_LX430={X 1291.24805,Y 1109.12805,Z 61.5505905,A -0.626630723,B 38.7113304,C -90.0650787,S 2,T 2,E1 6193.23291,E2 0.0,E3 0.0,E4 0.0,E5 0.0,E6 0.0}
DECL FDAT FXs_lx430={TOOL_NO 1,BASE_NO 1,IPO_FRAME #BASE,POINT2[] " ",TQ_STATE FALSE}
DECL E6POS XXS_LX431={X 1348.521,Y 1113.70105,Z 126.297096,A -0.588395178,B 1.75486195,C -90.0525818,S 2,T 2,E1 6075.11279,E2 0.0,E3 0.0,E4 0.0,E5 0.0,E6 0.0}
DECL FDAT FXs_lx431={TOOL_NO 1,BASE_NO 1,IPO_FRAME #BASE,POINT2[] " ",TQ_STATE FALSE}
DECL E6POS XXS_LX531={X 1273.10303,Y 1112.27405,Z 24.7617607,A -0.640370071,B 48.2600288,C -90.0756378,S 2,T 2,E1 6193.8999,E2 0.0,E3 0.0,E4 0.0,E5 0.0,E6 0.0}
DECL FDAT FXs_lx531={TOOL_NO 1,BASE_NO 1,IPO_FRAME #BASE,POINT2[] " ",TQ_STATE FALSE}
DECL PDAT PPDAT35={VEL 100.0,ACC 100.0,APO_DIST 20.0,APO_MODE #CDIS}
DECL E6POS XXS_LX532={X 1273.09595,Y 1106.79504,Z 52.060009,A -0.639810324,B 48.2610283,C -90.0751572,S 2,T 2,E1 6194.7832,E2 0.0,E3 0.0,E4 0.0,E5 0.0,E6 0.0}
DECL FDAT FXs_lx532={TOOL_NO 1,BASE_NO 1,IPO_FRAME #BASE,POINT2[] " ",TQ_STATE FALSE}
DECL PDAT PPDAT36={VEL 100.0,ACC 100.0,APO_DIST 20.0,APO_MODE #CDIS}
DECL E6POS XXS_LX421={X 1331.45801,Y 1113.62903,Z 140.508896,A -0.564055204,B -2.25771308,C -90.0505371,S 2,T 2,E1 5568.8999,E2 0.0,E3 0.0,E4 0.0,E5 0.0,E6 0.0}
DECL FDAT FXs_lx421={TOOL_NO 1,BASE_NO 1,IPO_FRAME #BASE,POINT2[] " ",TQ_STATE FALSE}
DECL E6POS XXS_LX422={X 1331.448,Y 1113.62598,Z 140.487,A -0.555783629,B -11.4802704,C -90.0506668,S 2,T 2,E1 5571.7002,E2 0.0,E3 0.0,E4 0.0,E5 0.0,E6 0.0}
DECL FDAT FXs_lx422={TOOL_NO 1,BASE_NO 1,IPO_FRAME #BASE,POINT2[] " ",TQ_STATE FALSE}
DECL E6POS XXS_LX534={X 1299.18005,Y 1113.90601,Z 155.308502,A -0.544914484,B -21.6417103,C -90.0528717,S 2,T 2,E1 5573.82813,E2 0.0,E3 0.0,E4 0.0,E5 0.0,E6 0.0}
DECL FDAT FXs_lx534={TOOL_NO 1,BASE_NO 1,IPO_FRAME #BASE,POINT2[] " ",TQ_STATE FALSE}
DECL PDAT PPDAT38={VEL 100.0,ACC 100.0,APO_DIST 100.0,APO_MODE #CDIS}
DECL E6POS XXS_LX423={X 1306.81396,Y 1263.76501,Z 115.999001,A -0.54406321,B -21.6427498,C -90.0545502,S 2,T 2,E1 5568.5918,E2 0.0,E3 0.0,E4 0.0,E5 0.0,E6 0.0}
DECL FDAT FXs_lx423={TOOL_NO 1,BASE_NO 1,IPO_FRAME #BASE,POINT2[] " ",TQ_STATE FALSE}
DECL E6POS XXS_LX424={X 1320.97205,Y 1519.14905,Z 108.012299,A 3.05467892,B -22.00144,C -89.1234894,S 2,T 2,E1 5572.271,E2 0.0,E3 0.0,E4 0.0,E5 0.0,E6 0.0}
DECL FDAT FXs_lx424={TOOL_NO 1,BASE_NO 1,IPO_FRAME #BASE,POINT2[] " ",TQ_STATE FALSE}
DECL E6POS XXS_LX535={X 1198.70996,Y 2189.93896,Z 25.40662,A -20.8274899,B -45.1372185,C -39.3026886,S 2,T 2,E1 5081.13379,E2 0.0,E3 0.0,E4 0.0,E5 0.0,E6 0.0}
DECL FDAT FXs_lx535={TOOL_NO 1,BASE_NO 1,IPO_FRAME #BASE,POINT2[] " ",TQ_STATE FALSE}
DECL PDAT PPDAT39={VEL 100.0,ACC 100.0,APO_DIST 100.0,APO_MODE #CDIS}
DECL E6POS XXS_LX537={X -459.137207,Y 2830.60693,Z -400.969299,A -93.8874512,B -1.00689602,C -1.81860495,S 2,T 2,E1 3742.04102,E2 0.0,E3 0.0,E4 0.0,E5 0.0,E6 0.0}
DECL FDAT FXs_lx537={TOOL_NO 1,BASE_NO 1,IPO_FRAME #BASE,POINT2[] " ",TQ_STATE FALSE}
DECL PDAT PPDAT41={VEL 100.0,ACC 100.0,APO_DIST 100.0,APO_MODE #CDIS}
DECL E6POS XXS_LX386={X -5394.59424,Y 2817.8999,Z -52.6045113,A -87.9566803,B 0.248233899,C 10.3403301,S 2,T 2,E1 -351.032715,E2 0.0,E3 0.0,E4 0.0,E5 0.0,E6 0.0}
DECL FDAT FXs_lx386={TOOL_NO 1,BASE_NO 1,IPO_FRAME #BASE,POINT2[] " ",TQ_STATE FALSE}
DECL SPOT_SUGG_T LAST_SPOT={GUN[] "1                       ",RETR_CMD[] "#CLO                    ",CHOISE[] "#FIRST                  ",CLO_TM[] "1                       ",PGNO1[] "25                      ",PRESS1[] "0                       ",PGNO2[] "1                       ",PRESS2[] "0                       ",SPOT_PARAMS[] "NORMAL                  "}
DECL PDAT PPDAT45={VEL 100.0,ACC 100.0,APO_DIST 100.0}
DECL E6POS XXS_LX546={X -1347.76294,Y 876.430298,Z -504.167694,A 136.986801,B 12.0716896,C -14.1013803,S 2,T 10,E1 4060.2981,E2 0.0,E3 0.0,E4 0.0,E5 0.0,E6 0.0}
DECL FDAT FXs_lx546={TOOL_NO 1,BASE_NO 1,IPO_FRAME #BASE,POINT2[] " ",TQ_STATE FALSE}
DECL PDAT PPDAT51={VEL 100.0,ACC 100.0,APO_DIST 100.0,APO_MODE #CDIS}
DECL E6POS XXS_LX548={X -1567.92603,Y 1474.04395,Z -380.613098,A -176.587601,B 10.73598,C -5.45803499,S 2,T 10,E1 4060.2981,E2 0.0,E3 0.0,E4 0.0,E5 0.0,E6 0.0}
DECL FDAT FXs_lx548={TOOL_NO 1,BASE_NO 1,IPO_FRAME #BASE,POINT2[] " ",TQ_STATE FALSE}
DECL PDAT PPDAT53={VEL 100.0,ACC 100.0,APO_DIST 100.0}
DECL E6POS XXS_LX463={X -285.360809,Y 775.312988,Z 375.377014,A -91.1736984,B -86.1419373,C 91.3704376,S 2,T 42,E1 4059.50293,E2 0.0,E3 0.0,E4 0.0,E5 0.0,E6 0.0}
DECL FDAT FXs_lx463={TOOL_NO 1,BASE_NO 1,IPO_FRAME #BASE,POINT2[] " ",TQ_STATE FALSE}
DECL E6POS XXS_LX552={X -7591.26416,Y 3233.35889,Z -215.513107,A -30.6375008,B 9.25732231,C -0.711479485,S 2,T 11,E1 -353.282715,E2 0.0,E3 0.0,E4 0.0,E5 0.0,E6 0.0}
DECL FDAT FXs_lx552={TOOL_NO 1,BASE_NO 1,IPO_FRAME #BASE,POINT2[] " ",TQ_STATE FALSE}
DECL PDAT PPDAT57={VEL 100.0,ACC 100.0,APO_DIST 100.0,APO_MODE #CDIS}
DECL PDAT PP_OLP116={VEL 100.0,ACC 100.0,APO_DIST 100.0,APO_MODE #CDIS}
DECL E6POS Xc_lx33={X -5797.43311,Y 2784.89893,Z -341.750305,A -179.385498,B 9.2559042,C -0.711720884,S 2,T 10,E1 -353.282196,E2 0.0,E3 0.0,E4 0.0,E5 0.0,E6 0.0}
DECL FDAT Fc_lx33={TOOL_NO 1,BASE_NO 2,IPO_FRAME #BASE,POINT2[] " ",TQ_STATE FALSE}
DECL E6POS XP2={X -1008.41998,Y -3878.53809,Z 2280.71802,A 15.8486004,B 69.8013687,C 116.1772,S 2,T 10,E1 3309.09106,E2 0.0,E3 0.0,E4 0.0,E5 0.0,E6 0.0}
DECL FDAT FP2={TOOL_NO 8,BASE_NO 0,IPO_FRAME #BASE,POINT2[] " ",TQ_STATE FALSE}
DECL PDAT PPDAT58={VEL 100.0,ACC 100.0,APO_DIST 100.0}
DECL E6POS XP3={X -2899.04102,Y 3376.81909,Z 87.3140106,A -134.810806,B 53.134861,C -12.8320503,S 2,T 10,E1 2156.50293,E2 0.0,E3 0.0,E4 0.0,E5 0.0,E6 0.0}
DECL FDAT FP3={TOOL_NO 1,BASE_NO 2,IPO_FRAME #BASE,POINT2[] " ",TQ_STATE FALSE}
DECL PDAT PPDAT59={VEL 100.0,ACC 100.0,APO_DIST 100.0,APO_MODE #CDIS}
DECL E6POS XXS_LX472={X -406.190887,Y 292.545807,Z -34.1930313,A 73.3883972,B -43.3940392,C -82.1220627,S 2,T 10,E1 4060.30005,E2 0.0,E3 0.0,E4 0.0,E5 0.0,E6 0.0}
DECL FDAT FXs_lx472={TOOL_NO 1,BASE_NO 1,IPO_FRAME #BASE,POINT2[] " ",TQ_STATE FALSE}
DECL E6POS XXS_LX443={X 490.55899,Y 1425.50195,Z -219.291702,A -179.175095,B -0.318304598,C 84.957428,S 2,T 34,E1 5250.30322,E2 0.0,E3 0.0,E4 0.0,E5 0.0,E6 0.0}
DECL FDAT FXs_lx443={TOOL_NO 1,BASE_NO 1,IPO_FRAME #BASE,POINT2[] " ",TQ_STATE FALSE}
DECL E6POS XXS_LX437={X 735.744385,Y 1314.55798,Z -205.183502,A -177.910797,B -6.01889086,C 78.0020905,S 2,T 34,E1 5254.11084,E2 0.0,E3 0.0,E4 0.0,E5 0.0,E6 0.0}
DECL FDAT FXs_lx437={TOOL_NO 1,BASE_NO 1,IPO_FRAME #BASE,POINT2[] " ",TQ_STATE FALSE}
DECL E6POS XXS_LX435={X 1247.71399,Y 1296.47705,Z -102.5009,A -0.543420196,B -50.1155205,C -90.0,S 2,T 2,E1 5252.6582,E2 0.0,E3 0.0,E4 0.0,E5 0.0,E6 0.0}
DECL FDAT FXs_lx435={TOOL_NO 1,BASE_NO 1,IPO_FRAME #BASE,POINT2[] " ",TQ_STATE FALSE}
DECL E6POS XXS_LX467={X 171.180801,Y 983.950684,Z -233.371597,A 68.1400681,B -45.7760887,C -90.0009766,S 2,T 10,E1 4060.30103,E2 0.0,E3 0.0,E4 0.0,E5 0.0,E6 0.0}
DECL FDAT FXs_lx467={TOOL_NO 1,BASE_NO 1,IPO_FRAME #BASE,POINT2[] " ",TQ_STATE FALSE}
DECL E6POS XXLX511={X 202.229294,Y 896.270508,Z 253.845901,A 90.3564911,B 13.9303102,C -88.6880264,S 2,T 10,E1 4060.302,E2 0.0,E3 0.0,E4 0.0,E5 0.0,E6 0.0}
DECL FDAT FXlx511={TOOL_NO 1,BASE_NO 1,IPO_FRAME #BASE,POINT2[] " ",TQ_STATE FALSE}
DECL E6POS XXLX509={X 162.742096,Y 891.286621,Z 202.198807,A 89.3670578,B 33.9861488,C -91.2537766,S 2,T 10,E1 4060.302,E2 0.0,E3 0.0,E4 0.0,E5 0.0,E6 0.0}
DECL FDAT FXlx509={TOOL_NO 1,BASE_NO 1,IPO_FRAME #BASE,POINT2[] " ",TQ_STATE FALSE}
DECL PDAT PP_OLP118={VEL 100.0,ACC 100.0,APO_DIST 100.0,APO_MODE #CDIS}
DECL E6POS XXs_lx464={X 166.837997,Y 775.260925,Z 368.354614,A -91.1741104,B -86.1427383,C 91.370903,S 2,T 42,E1 4058.85107,E2 0.0,E3 0.0,E4 0.0,E5 0.0,E6 0.0}
DECL FDAT FXs_lx464={TOOL_NO 1,BASE_NO 1,IPO_FRAME #BASE,POINT2[] " ",TQ_STATE FALSE}
DECL PDAT PP_OLP119={VEL 100.0,ACC 100.0,APO_DIST 0.0}
DECL E6POS Xswp_60_5097={X 155.421204,Y 677.644409,Z 419.4534,A -89.9986191,B -76.7324066,C 89.9989395,S 2,T 42,E1 4060.29907,E2 0.0,E3 0.0,E4 0.0,E5 0.0,E6 0.0}
DECL FDAT Fswp_60_5097={TOOL_NO 1,BASE_NO 1,IPO_FRAME #BASE,POINT2[] " "}
DECL PDAT PP_OLP120={VEL 100.0,ACC 100.0,APO_DIST 0.0}
DECL E6POS Xswp_60_5099={X 155.171906,Y 756.641907,Z 420.422699,A 24.4609909,B -89.997139,C -24.46138,S 2,T 42,E1 4060.29907,E2 0.0,E3 0.0,E4 0.0,E5 0.0,E6 0.0}
DECL FDAT Fswp_60_5099={TOOL_NO 1,BASE_NO 1,IPO_FRAME #BASE,POINT2[] " "}
DECL PDAT PP_OLP121={VEL 100.0,ACC 100.0,APO_DIST 0.0}
DECL E6POS Xswp_60_5101={X 155.733994,Y 840.013794,Z 421.443298,A 24.8737907,B -89.9972229,C -24.8741093,S 2,T 42,E1 4060.29907,E2 0.0,E3 0.0,E4 0.0,E5 0.0,E6 0.0}
DECL FDAT Fswp_60_5101={TOOL_NO 1,BASE_NO 1,IPO_FRAME #BASE,POINT2[] " "}
DECL PDAT PP_OLP122={VEL 100.0,ACC 100.0,APO_DIST 0.0}
DECL E6POS Xswp_60_5085={X 156.082306,Y 894.531006,Z 254.542404,A 89.7875671,B 15.1001301,C -91.0752563,S 2,T 10,E1 4060.30103,E2 0.0,E3 0.0,E4 0.0,E5 0.0,E6 0.0}
DECL FDAT Fswp_60_5085={TOOL_NO 1,BASE_NO 1,IPO_FRAME #BASE,POINT2[] " "}
DECL E6POS XP8={X -291.032288,Y 1013.00403,Z -302.712006,A -102.734497,B 68.9540329,C 77.207077,S 2,T 10,E1 4060.31104,E2 0.0,E3 0.0,E4 0.0,E5 0.0,E6 0.0}
DECL FDAT FP8={TOOL_NO 1,BASE_NO 1,IPO_FRAME #BASE,POINT2[] " ",TQ_STATE FALSE}
DECL PDAT PPDAT65={VEL 100.0,ACC 100.0,APO_DIST 100.0,APO_MODE #CDIS}
DECL E6POS XP9={X -205.798492,Y 207.417007,Z 211.056396,A -93.6165237,B 13.9594002,C 90.2877808,S 2,T 10,E1 4060.31104,E2 0.0,E3 0.0,E4 0.0,E5 0.0,E6 0.0}
DECL FDAT FP9={TOOL_NO 1,BASE_NO 1,IPO_FRAME #BASE,POINT2[] " ",TQ_STATE FALSE}
DECL PDAT PPDAT66={VEL 100.0,ACC 100.0,APO_DIST 100.0,APO_MODE #CDIS}
DECL E6POS XP10={X 190.3022,Y 135.982407,Z 204.456207,A -96.1434937,B 14.1406603,C 89.6691132,S 2,T 10,E1 4060.31201,E2 0.0,E3 0.0,E4 0.0,E5 0.0,E6 0.0}
DECL FDAT FP10={TOOL_NO 1,BASE_NO 1,IPO_FRAME #BASE,POINT2[] " ",TQ_STATE FALSE}
DECL PDAT PPDAT67={VEL 100.0,ACC 100.0,APO_DIST 100.0,APO_MODE #CDIS}
DECL PDAT PPDAT68={VEL 100.0,ACC 100.0,APO_DIST 100.0}
DECL E6POS XP13={X 169.981796,Y 176.841797,Z 220.672104,A -89.7854614,B 11.5515804,C 87.9993362,S 2,T 10,E1 4060.31494,E2 0.0,E3 0.0,E4 0.0,E5 0.0,E6 0.0}
DECL FDAT FP13={TOOL_NO 1,BASE_NO 1,IPO_FRAME #BASE,POINT2[] " ",TQ_STATE FALSE}
DECL PDAT PPDAT70={VEL 100.0,ACC 100.0,APO_DIST 100.0,APO_MODE #CDIS}
DECL PDAT PPDAT71={VEL 100.0,ACC 100.0,APO_DIST 100.0}
DECL PDAT PPDAT72={VEL 100.0,ACC 100.0,APO_DIST 100.0,APO_MODE #CDIS}
DECL E6POS Xpt1={X 161.814499,Y 201.080795,Z 274.221313,A -88.7676163,B -26.3682098,C 88.4874115,S 2,T 10,E1 4060.31494,E2 0.0,E3 0.0,E4 0.0,E5 0.0,E6 0.0}
DECL FDAT Fpt1={TOOL_NO 1,BASE_NO 1,IPO_FRAME #BASE,POINT2[] " ",TQ_STATE FALSE}
DECL PDAT PPDAT73={VEL 100.0,ACC 100.0,APO_DIST 100.0}
DECL E6POS XPT2={X 159.854294,Y 242.701508,Z 357.2724,A -87.5249329,B -56.4212418,C 88.3794632,S 2,T 10,E1 4060.31592,E2 0.0,E3 0.0,E4 0.0,E5 0.0,E6 0.0}
DECL FDAT Fpt2={TOOL_NO 1,BASE_NO 1,IPO_FRAME #BASE,POINT2[] " ",TQ_STATE FALSE}
DECL PDAT PPDAT74={VEL 100.0,ACC 100.0,APO_DIST 100.0,APO_MODE #CDIS}
DECL E6POS XPT3={X 169.334305,Y 358.47821,Z 399.365112,A 87.187088,B -69.8794937,C -84.8208008,S 2,T 10,E1 4060.31592,E2 0.0,E3 0.0,E4 0.0,E5 0.0,E6 0.0}
DECL FDAT Fpt3={TOOL_NO 1,BASE_NO 1,IPO_FRAME #BASE,POINT2[] " ",TQ_STATE FALSE}
DECL PDAT PPDAT75={VEL 100.0,ACC 100.0,APO_DIST 100.0,APO_MODE #CDIS}
DECL PDAT PPDAT76={VEL 100.0,ACC 100.0,APO_DIST 100.0}
DECL E6POS XPT4={X 163.896896,Y 440.960114,Z 374.004089,A 88.4197922,B -54.7953987,C -86.9808578,S 2,T 10,E1 4060.31299,E2 0.0,E3 0.0,E4 0.0,E5 0.0,E6 0.0}
DECL FDAT Fpt4={TOOL_NO 1,BASE_NO 1,IPO_FRAME #BASE,POINT2[] " ",TQ_STATE FALSE}
DECL PDAT PPDAT77={VEL 100.0,ACC 100.0,APO_DIST 100.0}
DECL E6POS XPT5={X -312.486206,Y 433.580505,Z 388.477386,A 88.4197922,B -54.7953987,C -86.9808578,S 2,T 10,E1 4060.31299,E2 0.0,E3 0.0,E4 0.0,E5 0.0,E6 0.0}
DECL FDAT Fpt5={TOOL_NO 1,BASE_NO 1,IPO_FRAME #BASE,POINT2[] " ",TQ_STATE FALSE}
DECL PDAT PPDAT78={VEL 100.0,ACC 100.0,APO_DIST 100.0,APO_MODE #CDIS}
DECL E6POS XPT6={X -312.831299,Y 431.701508,Z 162.645004,A 96.246109,B 71.9801483,C -84.3668823,S 2,T 10,E1 4060.31299,E2 0.0,E3 0.0,E4 0.0,E5 0.0,E6 0.0}
DECL FDAT Fpt6={TOOL_NO 1,BASE_NO 1,IPO_FRAME #BASE,POINT2[] " ",TQ_STATE FALSE}
DECL PDAT PPDAT79={VEL 100.0,ACC 100.0,APO_DIST 100.0,APO_MODE #CDIS}
DECL E6POS XPT7={X 154.929993,Y 439.048096,Z 148.423401,A 93.5119171,B 56.3998604,C -86.8548965,S 2,T 10,E1 4060.30005,E2 0.0,E3 0.0,E4 0.0,E5 0.0,E6 0.0}
DECL FDAT Fpt7={TOOL_NO 1,BASE_NO 1,IPO_FRAME #BASE,POINT2[] " ",TQ_STATE FALSE}
DECL PDAT PPDAT80={VEL 100.0,ACC 100.0,APO_DIST 100.0,APO_MODE #CDIS}
DECL E6POS XSWP_60_5209={X 156.664795,Y 490.26001,Z 142.292603,A 93.5122604,B 56.3994598,C -86.8546371,S 2,T 10,E1 4060.30005,E2 0.0,E3 0.0,E4 0.0,E5 0.0,E6 0.0}
DECL FDAT Fswp_60_5209={TOOL_NO 1,BASE_NO 1,IPO_FRAME #BASE,POINT2[] " ",TQ_STATE FALSE}
DECL PDAT PPDAT81={VEL 100.0,ACC 100.0,APO_DIST 100.0}
DECL PDAT PPDAT82={VEL 100.0,ACC 100.0,APO_DIST 100.0}
DECL E6POS Xpt8={X 154.929993,Y 439.048096,Z 148.423401,A 93.5119171,B 56.3998604,C -86.8548965,S 2,T 10,E1 4060.30005,E2 0.0,E3 0.0,E4 0.0,E5 0.0,E6 0.0}
DECL FDAT Fpt8={TOOL_NO 1,BASE_NO 1,IPO_FRAME #BASE,POINT2[] " ",TQ_STATE FALSE}
DECL E6POS XPT9={X -312.831299,Y 431.701508,Z 162.645004,A 96.246109,B 71.9801483,C -84.3668823,S 2,T 10,E1 4060.31299,E2 0.0,E3 0.0,E4 0.0,E5 0.0,E6 0.0}
DECL FDAT Fpt9={TOOL_NO 1,BASE_NO 1,IPO_FRAME #BASE,POINT2[] " ",TQ_STATE FALSE}
DECL PDAT PPDAT83={VEL 100.0,ACC 100.0,APO_DIST 100.0}
DECL E6POS XPT11={X 160.858307,Y 725.869202,Z 118.343903,A -89.463562,B 67.0390701,C 92.8514862,S 2,T 10,E1 4060.30396,E2 0.0,E3 0.0,E4 0.0,E5 0.0,E6 0.0}
DECL FDAT Fpt11={TOOL_NO 1,BASE_NO 1,IPO_FRAME #BASE,POINT2[] " ",TQ_STATE FALSE}
DECL PDAT PPDAT85={VEL 100.0,ACC 100.0,APO_DIST 100.0,APO_MODE #CDIS}
DECL E6POS XPT12={X 161.1828,Y 693.768921,Z 161.033401,A -90.1003571,B 49.8515396,C 94.0767822,S 2,T 10,E1 4060.30396,E2 0.0,E3 0.0,E4 0.0,E5 0.0,E6 0.0}
DECL FDAT Fpt12={TOOL_NO 1,BASE_NO 1,IPO_FRAME #BASE,POINT2[] " ",TQ_STATE FALSE}
DECL PDAT PPDAT86={VEL 100.0,ACC 100.0,APO_DIST 100.0,APO_MODE #CDIS}
DECL E6POS XPT13={X 175.753799,Y 675.288574,Z 178.158401,A -90.3979263,B 47.0033798,C 94.2010193,S 2,T 10,E1 4060.30493,E2 0.0,E3 0.0,E4 0.0,E5 0.0,E6 0.0}
DECL FDAT Fpt13={TOOL_NO 1,BASE_NO 1,IPO_FRAME #BASE,POINT2[] " ",TQ_STATE FALSE}
DECL PDAT PPDAT87={VEL 100.0,ACC 100.0,APO_DIST 100.0,APO_MODE #CDIS}
DECL E6POS XPT14={X 179.009003,Y 617.818115,Z 251.7612,A -92.1164398,B 18.5910301,C 93.9508972,S 2,T 10,E1 4060.30493,E2 0.0,E3 0.0,E4 0.0,E5 0.0,E6 0.0}
DECL FDAT Fpt14={TOOL_NO 1,BASE_NO 1,IPO_FRAME #BASE,POINT2[] " ",TQ_STATE FALSE}
DECL PDAT PPDAT88={VEL 100.0,ACC 100.0,APO_DIST 100.0,APO_MODE #CDIS}
DECL PDAT PPDAT89={VEL 100.0,ACC 100.0,APO_DIST 100.0}
DECL E6POS XPT15={X 179.009003,Y 617.818115,Z 251.7612,A -92.1164398,B 18.5910301,C 93.9508972,S 2,T 10,E1 4060.30493,E2 0.0,E3 0.0,E4 0.0,E5 0.0,E6 0.0}
DECL FDAT Fpt15={TOOL_NO 1,BASE_NO 1,IPO_FRAME #BASE,POINT2[] " ",TQ_STATE FALSE}
DECL PDAT PPDAT90={VEL 100.0,ACC 100.0,APO_DIST 100.0}
DECL E6POS XPT16={X 175.753799,Y 675.288574,Z 178.158401,A -90.3979263,B 47.0033798,C 94.2010193,S 2,T 10,E1 4060.30493,E2 0.0,E3 0.0,E4 0.0,E5 0.0,E6 0.0}
DECL FDAT Fpt16={TOOL_NO 1,BASE_NO 1,IPO_FRAME #BASE,POINT2[] " ",TQ_STATE FALSE}
DECL PDAT PPDAT91={VEL 100.0,ACC 100.0,APO_DIST 100.0,APO_MODE #CDIS}
DECL E6POS XPT18={X 161.1828,Y 693.768921,Z 161.033401,A -90.1003571,B 49.8515396,C 94.0767822,S 2,T 10,E1 4060.30396,E2 0.0,E3 0.0,E4 0.0,E5 0.0,E6 0.0}
DECL FDAT Fpt18={TOOL_NO 1,BASE_NO 1,IPO_FRAME #BASE,POINT2[] " ",TQ_STATE FALSE}
DECL PDAT PPDAT93={VEL 100.0,ACC 100.0,APO_DIST 100.0,APO_MODE #CDIS}
DECL E6POS XPT19={X 160.822693,Y 729.790894,Z 127.590401,A -89.4637833,B 67.0392914,C 92.8511581,S 2,T 10,E1 4060.30396,E2 0.0,E3 0.0,E4 0.0,E5 0.0,E6 0.0}
DECL FDAT Fpt19={TOOL_NO 1,BASE_NO 1,IPO_FRAME #BASE,POINT2[] " ",TQ_STATE FALSE}
DECL PDAT PPDAT94={VEL 100.0,ACC 100.0,APO_DIST 100.0,APO_MODE #CDIS}
DECL E6POS XPT20={X 217.4048,Y 2369.823,Z -30.3654709,A -73.5321121,B -28.8238201,C -1.98111796,S 2,T 2,E1 4846.66211,E2 0.0,E3 0.0,E4 0.0,E5 0.0,E6 0.0}
DECL FDAT Fpt20={TOOL_NO 1,BASE_NO 1,IPO_FRAME #BASE,POINT2[] " ",TQ_STATE FALSE}
DECL PDAT PPDAT95={VEL 100.0,ACC 100.0,APO_DIST 100.0,APO_MODE #CDIS}
DECL E6POS XP14={X 673.541199,Y 1727.53601,Z 1378.01599,A 0.981028795,B -89.2553635,C -78.1354065,S 2,T 2,E1 5254.5,E2 0.0,E3 0.0,E4 0.0,E5 0.0,E6 0.0}
DECL FDAT FP14={TOOL_NO 1,BASE_NO 1,IPO_FRAME #BASE,POINT2[] " ",TQ_STATE FALSE}
DECL PDAT PPDAT96={VEL 100.0,ACC 100.0,APO_DIST 100.0,APO_MODE #CDIS}
DECL E6POS XP15={X 373.471985,Y 1712.46106,Z 714.465271,A 159.352203,B -72.0383682,C 115.424301,S 2,T 2,E1 5255.12988,E2 0.0,E3 0.0,E4 0.0,E5 0.0,E6 0.0}
DECL FDAT FP15={TOOL_NO 1,BASE_NO 1,IPO_FRAME #BASE,POINT2[] " ",TQ_STATE FALSE}
DECL PDAT PPDAT97={VEL 100.0,ACC 100.0,APO_DIST 100.0,APO_MODE #CDIS}
ENDDAT
